RoboDK station: SetToolCutter wrt Tool Holder.rdk

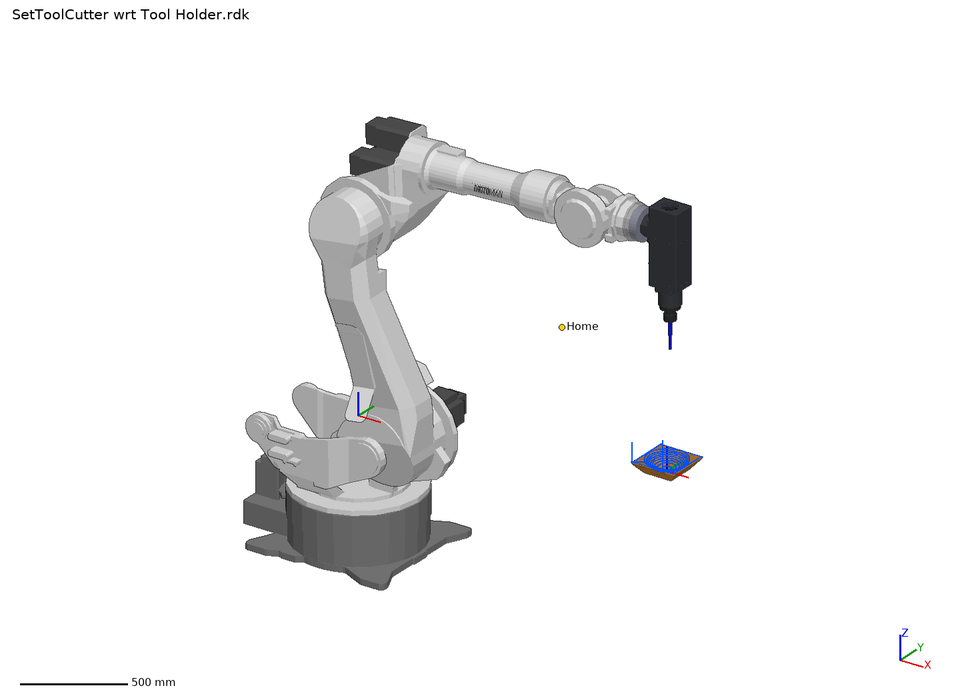
[picture v0: the station drawn from its stored meshes, robots at their saved joint values, targets as dots, program paths as lines]
Station Example Automatic Tool Cutters. Poses are relative to the parent item; angles as X-Y-Z fixed-axis rotations.
  - Python program SetToolCutter (listed below)
  - frame Motoman ES200D Base at (0, 0, 0) mm
    - robot Motoman ES200D: 6 axes, payload 200 kg, reach 2651 mm, repeatability 0.2 mm, weight 1130 kg
        modified DH rows (alpha deg, a mm, theta deg, d mm): 0, 0, 0, 650; -90, 285, -90, 0; 0, 1150, 0, 0; -90, 250, 0, 1225; 90, 0, 0, 0; -90, 0, 0, 250
        base shift (0, 0, -650) mm
        joint limits [-180, -60, -142.5, -360, -125, -360] to [180, 76, 230, 360, 125, 360]; home [0, 0, 0, 0, 0, 0]; saved at [0, -7.655, -4.967, 0, -2.688, 180]
      - tool Tool Holder, TCP at (456.22, 0, 176) mm, rotated rx 0 ry 90 rz 0 deg, size 592.9 x 170 x 256 mm
      - tool Tool 10-150, TCP at (606.22, 0, 176) mm, rotated rx 0 ry 90 rz 0 deg
        - object Cutter 10-150 at (0, 0, 0) mm, size 10 x 10 x 150 mm, geometry from Part.sld
      - tool Tool 20-75, TCP at (531.22, 0, 176) mm, rotated rx 0 ry 90 rz 0 deg
        - object Cutter 20-75 at (0, 0, 0) mm, size 20 x 20 x 75 mm, geometry from Part.sld
    - frame Milling Reference at (1817.19, -92.29, 260.27) mm
      - object Wooden bowl at (0, 0, 0) mm, size 241.3 x 241.3 x 60 mm
      - target Home (joint target) at (-659.05, 92.29, 521.01) mm, rotated rx 180 ry 0 rz -180 deg; joints [0, -37.94, -26.87, 0, -11.07, 180] of Motoman ES200D
  - machining project Machining Settings: Q:/RoboDK/Deploy/RoboDK_vc2013x64/Library/Milling 3axis bowl.nc | rotZ(0) | rotX(0)*rotY(0) | onStart | onPathStart | onApproach | onPoint | onRetract | onFinish | Extruder(%1) | default | default | OutOnMov(%1) | OutOffMov(%1) | onPathFinish | M_RunCode(%1)
  - program Machining (918 instructions, listed below)
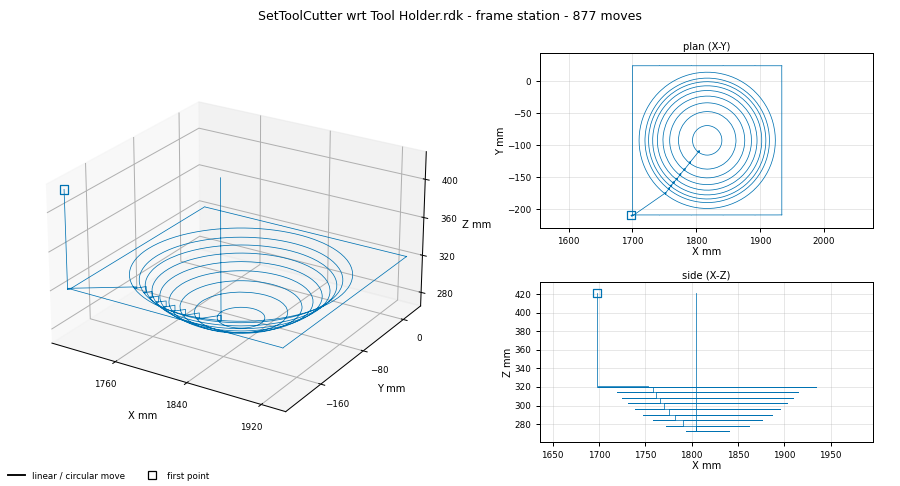
[picture p0: tool path of SetToolCutter wrt Tool Holder.rdk in frame station, 877 of 877 moves have a stored position in this frame; points joined in program order, loops and branches not executed]

--- Python program SetToolCutter ---
# This example shows how to programmatically select (and, if necessary, automatically create) a tool that does not exist
# This is meant to be used for robot machining projects where a tool holder is used as a reference tool
#
# Documentation: https://robodk.com/doc/en/RoboDK-API.html
# Reference:     https://robodk.com/doc/en/PythonAPI/index.html
# Note: It is not required to keep a copy of this file, your python script is saved with the station
from robolink import *    # RoboDK API
from robodk import *      # Robot toolbox
RDK = Robolink()

# Ask the user to select a tool holder
tool_holder = RDK.ItemUserPick('Select a the tool holder (TCP spindle reference)', ITEM_TYPE_TOOL)
# Alernatively, pick a named tool holder:
# tool_holder = RDK.Item('Tool Holder', ITEM_TYPE_TOOL)
# Or, the first tool of a robot:
# tool_holder = robot.Childs()[0]

# Exit if the tool does not exist
if not tool_holder.Valid():
    raise Exception("The tool holder was not selected")

# Retrieve the robot
robot = tool_holder.Parent()

# Ask the user to enter the tool parameters
user_input = mbox("Enter the tool diameter and length (in mm) using the following format:\ndiameter-length\n\nExample:\n10-150", entry="10-150")
if user_input is False:
    print("Operation cancelled")
    quit(0)

# Convert the string to diameter and length variables
diam_length = user_input.split('-')
try:
    diameter = float(diam_length[0])
    length = float(diam_length[1])
except:
    raise Exception("Invalid input: " + diam_length)

# Create a new tool and add the geometry to it
tool_i_name = 'Tool %s' % user_input
tool_i = RDK.Item(tool_i_name, ITEM_TYPE_TOOL)
if tool_i.Valid():
    print("The tool already exists")

else:
    # If the tool holder Z axis points towards the outsite:
    tool_i_pose = tool_holder.PoseTool() * transl(0,0,length)
    # If the tool holder Z axis points towards the inside:
    #tool_i_pose = tool_holder.PoseTool() * transl(0,0,length) * rotx(pi)
    tool_i = robot.AddTool(tool_i_pose, tool_i_name)

    # RoboDK library comes with a sample part that always has the same name
    # this Part.sld is 80 mm in diameter and 100 mm long
    tool1_shape = RDK.AddFile(RDK.getParam('PATH_LIBRARY') + '/Part.sld', tool_i)
    tool1_shape.setName("Cutter %s" % user_input)
    tool1_shape.setGeometryPose(rotx(pi))
    # Scale the object accordingly
    tool1_shape.Scale([ diameter/60,   diameter/60,   length/80  ])
    # Change the color
    tool1_shape.Recolor([0,0,1,0.4]) # make the drill bit blue & transparent (RGBA): if transparency is under 80% it won't check for collisions (when you activate collision checking).


# Set the active tool
robot.setTool(tool_i)

--- program Machining (robot Motoman ES200D) ---
  Set Ref.: Milling Reference
  Set Tool: Tool 10-150
  Show Tool 10-150
  Set speed (1000.0 mm/s)
  Set speed (1000.0 mm/s)
  MoveJ 1 to (-119.55, -117.48, 161.2) mm, rotated rx 180 ry 0 rz 180 deg; joints [-9.367, -12.184, -28.14, -149.033, -18.441, -29.651]
  MoveL 2 to (-119.55, -117.48, 161.2) mm, rotated rx 180 ry 0 rz 180 deg; joints [-9.367, -12.184, -28.14, -149.033, -18.441, -29.651]
  MoveL 3 to (-119.55, -117.48, 61.2) mm, rotated rx -180 ry 0 rz 180 deg; joints [-9.367, -11.562, -32.254, -154.973, -22.628, -23.313]
  MoveL 4 to (-119.55, -117.48, 61.2) mm, rotated rx -180 ry 0 rz 180 deg; joints [-9.367, -11.562, -32.254, -154.973, -22.628, -23.313]
  Set speed (5.0 mm/s)
  MoveL 5 to (-119.55, -117.48, 60) mm, rotated rx -180 ry 0 rz -180 deg; joints [-9.367, -11.552, -32.301, -155.032, -22.68, -23.25]
  MoveL 6 to (-118.15, -118.45, 60) mm, rotated rx -180 ry 0 rz -180 deg; joints [-9.4, -11.471, -32.235, -154.97, -22.707, -23.304]
  MoveL 7 to (-117.59, -118.18, 60) mm, rotated rx -180 ry 0 rz -180 deg; joints [-9.384, -11.444, -32.213, -155.013, -22.705, -23.264]
  MoveL 8 to (-117.24, -117.67, 60) mm, rotated rx -180 ry 0 rz -180 deg; joints [-9.359, -11.43, -32.202, -155.075, -22.698, -23.206]
  MoveL 9 to (-117.19, -117.05, 60) mm, rotated rx -180 ry 0 rz 180 deg; joints [-9.331, -11.433, -32.204, -155.14, -22.686, -23.146]
  Set speed (16.7 mm/s)
  MoveL 10 to (-117.29, -116.49, 60) mm, rotated rx -180 ry 0 rz -180 deg; joints [-9.308, -11.443, -32.212, -155.194, -22.675, -23.096]
  MoveL 11 to (-116.89, -115.89, 60) mm, rotated rx 180 ry 0 rz 180 deg; joints [-9.278, -11.427, -32.2, -155.268, -22.666, -23.028]
  MoveL 12 to (-116.98, -83.97, 60) mm, rotated rx 180 ry 0 rz 180 deg; joints [-7.876, -11.682, -32.407, -158.649, -22.109, -19.909]
  MoveL 13 to (-116.98, 115.67, 60) mm, rotated rx 180 ry 0 rz 180 deg; joints [1.051, -12.311, -32.914, -182.985, -20.629, 2.794]
  MoveL 14 to (-117.29, 116.83, 60) mm, rotated rx 180 ry 0 rz 180 deg; joints [1.103, -12.326, -32.926, -183.133, -20.628, 2.933]
  MoveL 15 to (-117.05, 117.18, 60) mm, rotated rx 180 ry 0 rz 180 deg; joints [1.119, -12.313, -32.916, -183.177, -20.632, 2.974]
  MoveL 16 to (-116.46, 117.29, 60) mm, rotated rx -180 ry 0 rz 180 deg; joints [1.123, -12.282, -32.891, -183.189, -20.638, 2.985]
  MoveL 17 to (-115.99, 116.9, 60) mm, rotated rx -180 ry 0 rz -180 deg; joints [1.106, -12.257, -32.871, -183.137, -20.642, 2.936]
  MoveL 18 to (-110.81, 116.98, 60) mm, rotated rx 180 ry 0 rz 180 deg; joints [1.105, -11.984, -32.651, -183.127, -20.695, 2.926]
  MoveL 19 to (-75.63, 116.98, 60) mm, rotated rx -180 ry 0 rz -180 deg; joints [1.075, -10.139, -31.136, -182.998, -21.023, 2.799]
  MoveL 20 to (-75.08, 117.32, 60) mm, rotated rx 180 ry 0 rz -180 deg; joints [1.09, -10.111, -31.112, -183.038, -21.029, 2.836]
  MoveL 21 to (-74.41, 116.98, 60) mm, rotated rx 180 ry 0 rz 180 deg; joints [1.074, -10.076, -31.083, -182.994, -21.034, 2.795]
  MoveL 22 to (-25.6, 116.98, 60) mm, rotated rx -180 ry 0 rz -180 deg; joints [1.036, -7.548, -28.917, -182.84, -21.392, 2.645]
  MoveL 23 to (-25.06, 117.33, 60) mm, rotated rx -180 ry 0 rz 180 deg; joints [1.05, -7.52, -28.892, -182.879, -21.397, 2.681]
  MoveL 24 to (-24.38, 116.98, 60) mm, rotated rx 180 ry 0 rz 180 deg; joints [1.035, -7.486, -28.862, -182.837, -21.4, 2.642]
  MoveL 25 to (24.43, 116.98, 60) mm, rotated rx -180 ry 0 rz -180 deg; joints [0.999, -4.992, -26.621, -182.709, -21.651, 2.518]
  MoveL 26 to (24.88, 117.31, 60) mm, rotated rx 180 ry 0 rz -180 deg; joints [1.012, -4.969, -26.6, -182.743, -21.654, 2.55]
  MoveL 27 to (25.65, 116.98, 60) mm, rotated rx 180 ry 0 rz 180 deg; joints [0.998, -4.93, -26.564, -182.706, -21.656, 2.515]
  MoveL 28 to (74.35, 116.98, 60) mm, rotated rx 180 ry 0 rz 180 deg; joints [0.965, -2.47, -24.252, -182.599, -21.803, 2.413]
  MoveL 29 to (74.9, 117.32, 60) mm, rotated rx -180 ry 0 rz 180 deg; joints [0.978, -2.442, -24.226, -182.634, -21.805, 2.445]
  MoveL 30 to (75.57, 116.98, 60) mm, rotated rx -180 ry 0 rz -180 deg; joints [0.964, -2.408, -24.193, -182.597, -21.805, 2.411]
  MoveL 31 to (115.94, 116.98, 60) mm, rotated rx 180 ry 0 rz 180 deg; joints [0.938, -0.388, -22.219, -182.522, -21.85, 2.341]
  MoveL 32 to (116.4, 117.29, 60) mm, rotated rx 180 ry 0 rz 180 deg; joints [0.95, -0.365, -22.196, -182.553, -21.851, 2.37]
  MoveL 33 to (116.91, 117.27, 60) mm, rotated rx 180 ry 0 rz 180 deg; joints [0.949, -0.339, -22.171, -182.55, -21.851, 2.367]
  MoveL 34 to (117.31, 116.72, 60) mm, rotated rx -180 ry 0 rz -180 deg; joints [0.928, -0.32, -22.151, -182.494, -21.85, 2.315]
  MoveL 35 to (117.11, 116.16, 60) mm, rotated rx -180 ry 0 rz -180 deg; joints [0.907, -0.33, -22.162, -182.437, -21.849, 2.262]
  MoveL 36 to (116.89, 115.69, 60) mm, rotated rx -180 ry 0 rz -180 deg; joints [0.889, -0.341, -22.173, -182.389, -21.849, 2.218]
  MoveL 37 to (116.98, 83.78, 60) mm, rotated rx 180 ry 0 rz 180 deg; joints [-0.323, -0.345, -22.176, -179.13, -21.834, -0.807]
  MoveL 38 to (116.98, -115.86, 60) mm, rotated rx -180 ry 0 rz -180 deg; joints [-7.858, 0.366, -21.465, -159.638, -23.137, -18.844]
  MoveL 39 to (117.33, -116.64, 60) mm, rotated rx -180 ry 0 rz -180 deg; joints [-7.885, 0.389, -21.443, -159.572, -23.146, -18.905]
  MoveL 40 to (117.02, -117.21, 60) mm, rotated rx -180 ry 0 rz 180 deg; joints [-7.908, 0.378, -21.454, -159.518, -23.153, -18.955]
  MoveL 41 to (116.53, -117.29, 60) mm, rotated rx 180 ry 0 rz 180 deg; joints [-7.914, 0.354, -21.478, -159.505, -23.155, -18.967]
  MoveL 42 to (115.95, -116.9, 60) mm, rotated rx -180 ry 0 rz -180 deg; joints [-7.902, 0.323, -21.509, -159.532, -23.152, -18.942]
  MoveL 43 to (110.78, -116.98, 60) mm, rotated rx -180 ry 0 rz 180 deg; joints [-7.932, 0.068, -21.764, -159.461, -23.162, -19.007]
  MoveL 44 to (75.6, -116.98, 60) mm, rotated rx -180 ry 0 rz -180 deg; joints [-8.12, -1.672, -23.482, -158.992, -23.203, -19.441]
  MoveL 45 to (75.05, -117.33, 60) mm, rotated rx -180 ry 0 rz -180 deg; joints [-8.136, -1.697, -23.506, -158.952, -23.208, -19.478]
  MoveL 46 to (74.38, -116.98, 60) mm, rotated rx -180 ry 0 rz -180 deg; joints [-8.127, -1.733, -23.541, -158.975, -23.203, -19.457]
  MoveL 47 to (25.57, -116.98, 60) mm, rotated rx -180 ry 0 rz -180 deg; joints [-8.403, -4.165, -25.856, -158.216, -23.188, -20.172]
  MoveL 48 to (25.02, -117.34, 60) mm, rotated rx -180 ry 0 rz 180 deg; joints [-8.42, -4.19, -25.879, -158.173, -23.193, -20.211]
  MoveL 49 to (24.35, -116.98, 60) mm, rotated rx -180 ry 0 rz -180 deg; joints [-8.41, -4.226, -25.913, -158.195, -23.187, -20.191]
  MoveL 50 to (-24.36, -116.98, 60) mm, rotated rx -180 ry 0 rz -180 deg; joints [-8.705, -6.679, -28.148, -157.299, -23.089, -21.048]
  MoveL 51 to (-25, -117.35, 60) mm, rotated rx -180 ry 0 rz -180 deg; joints [-8.724, -6.708, -28.174, -157.251, -23.093, -21.092]
  MoveL 52 to (-25.58, -116.98, 60) mm, rotated rx 180 ry 0 rz 180 deg; joints [-8.713, -6.74, -28.203, -157.275, -23.086, -21.071]
  MoveL 53 to (-74.39, -116.98, 60) mm, rotated rx -180 ry 0 rz 180 deg; joints [-9.03, -9.227, -30.367, -156.219, -22.907, -22.093]
  MoveL 54 to (-74.94, -117.33, 60) mm, rotated rx -180 ry 0 rz -180 deg; joints [-9.049, -9.252, -30.388, -156.171, -22.91, -22.137]
  MoveL 55 to (-75.61, -116.98, 60) mm, rotated rx 180 ry 0 rz 180 deg; joints [-9.038, -9.289, -30.42, -156.19, -22.901, -22.121]
  MoveL 56 to (-115.98, -116.98, 60) mm, rotated rx 180 ry 0 rz 180 deg; joints [-9.32, -11.371, -32.154, -155.179, -22.692, -23.108]
  MoveL 57 to (-116.63, -117.33, 60) mm, rotated rx -180 ry 0 rz -180 deg; joints [-9.34, -11.401, -32.179, -155.126, -22.695, -23.158]
  MoveL 58 to (-117.19, -117.05, 60) mm, rotated rx -180 ry 0 rz 180 deg; joints [-9.331, -11.433, -32.204, -155.14, -22.686, -23.146]
  Set speed (16.7 mm/s)
  MoveL 59 to (-117.8, -116.93, 60) mm, rotated rx 180 ry 0 rz 180 deg; joints [-9.33, -11.465, -32.231, -155.136, -22.68, -23.151]
  MoveL 60 to (-118.38, -117.12, 60) mm, rotated rx 180 ry 0 rz 180 deg; joints [-9.343, -11.494, -32.254, -155.1, -22.681, -23.185]
  MoveL 61 to (-118.8, -117.59, 60) mm, rotated rx 180 ry 0 rz -180 deg; joints [-9.367, -11.512, -32.268, -155.041, -22.687, -23.24]
  MoveL 62 to (-118.26, -119.2, 60) mm, rotated rx -180 ry 0 rz -180 deg; joints [-9.433, -11.47, -32.234, -154.89, -22.72, -23.378]
  MoveL 63 to (-118.26, -119.2, 61.2) mm, rotated rx 180 ry 0 rz 180 deg; joints [-9.433, -11.48, -32.187, -154.832, -22.668, -23.441]
  Set speed (1000.0 mm/s)
  MoveL 64 to (-64.77, -81.96, 61.2) mm, rotated rx -180 ry 0 rz 180 deg; joints [-7.484, -9.005, -30.122, -159.967, -22.347, -18.637]
  Set speed (5.0 mm/s)
  MoveL 65 to (-64.77, -81.96, 60) mm, rotated rx 180 ry 0 rz 180 deg; joints [-7.484, -8.994, -30.169, -160.014, -22.401, -18.585]
  MoveL 66 to (-66.46, -82.15, 60) mm, rotated rx 180 ry 0 rz 180 deg; joints [-7.502, -9.08, -30.242, -159.959, -22.395, -18.637]
  MoveL 67 to (-66.71, -82.72, 60) mm, rotated rx -180 ry 0 rz -180 deg; joints [-7.527, -9.088, -30.249, -159.895, -22.402, -18.697]
  MoveL 68 to (-66.64, -83.34, 60) mm, rotated rx 180 ry 0 rz 180 deg; joints [-7.553, -9.08, -30.242, -159.831, -22.411, -18.756]
  MoveL 69 to (-66.26, -83.84, 60) mm, rotated rx -180 ry 0 rz -180 deg; joints [-7.572, -9.058, -30.223, -159.787, -22.42, -18.796]
  Set speed (16.7 mm/s)
  MoveL 70 to (-60.03, -88.41, 60) mm, rotated rx -180 ry 0 rz -180 deg; joints [-7.731, -8.707, -29.922, -159.438, -22.519, -19.112]
  MoveL 71 to (-53.48, -92.52, 60) mm, rotated rx -180 ry 0 rz 180 deg; joints [-7.866, -8.342, -29.608, -159.148, -22.611, -19.373]
  MoveL 72 to (-46.6, -96.17, 60) mm, rotated rx -180 ry 0 rz -180 deg; joints [-7.979, -7.965, -29.281, -158.915, -22.695, -19.582]
  MoveL 73 to (-39.63, -99.24, 60) mm, rotated rx -180 ry 0 rz -180 deg; joints [-8.066, -7.587, -28.951, -158.743, -22.769, -19.733]
  MoveL 74 to (-32.34, -101.86, 60) mm, rotated rx -180 ry 0 rz 180 deg; joints [-8.131, -7.197, -28.607, -158.625, -22.835, -19.835]
  MoveL 75 to (-25.37, -103.8, 60) mm, rotated rx 180 ry 0 rz 180 deg; joints [-8.17, -6.829, -28.281, -158.567, -22.887, -19.883]
  MoveL 76 to (-25.08, -103.7, 60) mm, rotated rx 180 ry 0 rz 180 deg; joints [-8.164, -6.815, -28.269, -158.583, -22.886, -19.868]
  MoveL 77 to (-24.41, -104.03, 60) mm, rotated rx 180 ry 0 rz 180 deg; joints [-8.174, -6.779, -28.237, -158.563, -22.894, -19.886]
  MoveL 78 to (-20.17, -104.94, 60) mm, rotated rx -180 ry 0 rz -180 deg; joints [-8.186, -6.557, -28.039, -158.553, -22.92, -19.891]
  MoveL 79 to (-12.53, -106.13, 60) mm, rotated rx 180 ry 0 rz 180 deg; joints [-8.19, -6.162, -27.685, -158.58, -22.959, -19.861]
  MoveL 80 to (-4.79, -106.76, 60) mm, rotated rx 180 ry 0 rz 180 deg; joints [-8.17, -5.766, -27.328, -158.661, -22.988, -19.781]
  MoveL 81 to (2.85, -106.83, 60) mm, rotated rx -180 ry 0 rz 180 deg; joints [-8.129, -5.38, -26.977, -158.79, -23.007, -19.657]
  MoveL 82 to (10.59, -106.34, 60) mm, rotated rx -180 ry 0 rz 180 deg; joints [-8.065, -4.994, -26.623, -158.972, -23.016, -19.485]
  MoveL 83 to (18.23, -105.3, 60) mm, rotated rx -180 ry 0 rz -180 deg; joints [-7.981, -4.618, -26.276, -159.201, -23.016, -19.27]
  MoveL 84 to (24.4, -104.03, 60) mm, rotated rx -180 ry 0 rz -180 deg; joints [-7.896, -4.317, -25.997, -159.424, -23.008, -19.062]
  MoveL 85 to (24.95, -103.68, 60) mm, rotated rx 180 ry 0 rz 180 deg; joints [-7.879, -4.292, -25.974, -159.466, -23.004, -19.023]
  MoveL 86 to (25.37, -103.8, 60) mm, rotated rx -180 ry 0 rz -180 deg; joints [-7.881, -4.27, -25.953, -159.462, -23.007, -19.027]
  MoveL 87 to (32.05, -101.95, 60) mm, rotated rx -180 ry 0 rz 180 deg; joints [-7.772, -3.948, -25.653, -159.745, -22.991, -18.763]
  MoveL 88 to (39.3, -99.38, 60) mm, rotated rx 180 ry 0 rz 180 deg; joints [-7.631, -3.602, -25.328, -160.102, -22.967, -18.431]
  MoveL 89 to (46.36, -96.29, 60) mm, rotated rx -180 ry 0 rz 180 deg; joints [-7.473, -3.269, -25.015, -160.502, -22.935, -18.061]
  MoveL 90 to (53.22, -92.67, 60) mm, rotated rx 180 ry 0 rz 180 deg; joints [-7.297, -2.95, -24.711, -160.945, -22.896, -17.651]
  MoveL 91 to (59.78, -88.58, 60) mm, rotated rx -180 ry 0 rz -180 deg; joints [-7.106, -2.648, -24.423, -161.426, -22.852, -17.205]
  MoveL 92 to (65.97, -84.07, 60) mm, rotated rx 180 ry 0 rz 180 deg; joints [-6.901, -2.367, -24.154, -161.939, -22.803, -16.731]
  MoveL 93 to (71.86, -79.09, 60) mm, rotated rx -180 ry 0 rz 180 deg; joints [-6.681, -2.103, -23.899, -162.49, -22.75, -16.222]
  MoveL 94 to (74.29, -76.81, 60) mm, rotated rx 180 ry 0 rz 180 deg; joints [-6.582, -1.995, -23.795, -162.739, -22.726, -15.992]
  MoveL 95 to (74.58, -76.19, 60) mm, rotated rx 180 ry 0 rz 180 deg; joints [-6.557, -1.984, -23.784, -162.802, -22.719, -15.934]
  MoveL 96 to (75.15, -75.96, 60) mm, rotated rx -180 ry 0 rz -180 deg; joints [-6.546, -1.957, -23.758, -162.831, -22.717, -15.907]
  MoveL 97 to (80.34, -70.47, 60) mm, rotated rx -180 ry 0 rz 180 deg; joints [-6.312, -1.729, -23.537, -163.42, -22.66, -15.363]
  MoveL 98 to (85.23, -64.46, 60) mm, rotated rx -180 ry 0 rz -180 deg; joints [-6.061, -1.518, -23.332, -164.054, -22.6, -14.777]
  MoveL 99 to (89.66, -58.15, 60) mm, rotated rx 180 ry 0 rz 180 deg; joints [-5.801, -1.33, -23.148, -164.712, -22.54, -14.169]
  MoveL 100 to (93.63, -51.52, 60) mm, rotated rx -180 ry 0 rz 180 deg; joints [-5.532, -1.165, -22.987, -165.396, -22.478, -13.537]
  MoveL 101 to (97.05, -44.73, 60) mm, rotated rx 180 ry 0 rz 180 deg; joints [-5.261, -1.027, -22.851, -166.09, -22.419, -12.896]
  MoveL 102 to (100.02, -37.64, 60) mm, rotated rx -180 ry 0 rz -180 deg; joints [-4.98, -0.911, -22.737, -166.81, -22.359, -12.23]
  MoveL 103 to (102.44, -30.41, 60) mm, rotated rx 180 ry 0 rz 180 deg; joints [-4.696, -0.82, -22.647, -167.541, -22.302, -11.553]
  MoveL 104 to (102.51, -30.2, 60) mm, rotated rx -180 ry 0 rz -180 deg; joints [-4.688, -0.818, -22.645, -167.562, -22.301, -11.533]
  MoveL 105 to (104.4, -22.82, 60) mm, rotated rx -180 ry 0 rz 180 deg; joints [-4.401, -0.753, -22.581, -168.305, -22.246, -10.846]
  MoveL 106 to (105.76, -15.32, 60) mm, rotated rx 180 ry 0 rz 180 deg; joints [-4.112, -0.713, -22.541, -169.058, -22.194, -10.149]
  MoveL 107 to (106.59, -7.67, 60) mm, rotated rx -180 ry 0 rz -180 deg; joints [-3.818, -0.698, -22.527, -169.824, -22.144, -9.439]
  MoveL 108 to (106.86, -0.29, 60) mm, rotated rx -180 ry 0 rz 180 deg; joints [-3.536, -0.709, -22.537, -170.563, -22.099, -8.755]
  MoveL 109 to (106.86, 0.23, 60) mm, rotated rx 180 ry 0 rz 180 deg; joints [-3.517, -0.71, -22.538, -170.615, -22.096, -8.706]
  MoveL 110 to (106.57, 7.9, 60) mm, rotated rx 180 ry 0 rz 180 deg; joints [-3.225, -0.747, -22.575, -171.383, -22.053, -7.995]
  MoveL 111 to (105.8, 14.83, 60) mm, rotated rx 180 ry 0 rz 180 deg; joints [-2.962, -0.804, -22.631, -172.077, -22.017, -7.352]
  MoveL 112 to (104.08, 24.16, 60) mm, rotated rx 180 ry 0 rz 180 deg; joints [-2.609, -0.913, -22.738, -173.013, -21.973, -6.484]
  MoveL 113 to (102.39, 30.57, 60) mm, rotated rx 180 ry 0 rz 180 deg; joints [-2.367, -1.011, -22.835, -173.656, -21.946, -5.887]
  MoveL 114 to (102.13, 31.4, 60) mm, rotated rx 180 ry 0 rz 180 deg; joints [-2.335, -1.026, -22.849, -173.741, -21.942, -5.809]
  MoveL 115 to (99.93, 37.84, 60) mm, rotated rx -180 ry 0 rz -180 deg; joints [-2.091, -1.148, -22.97, -174.389, -21.917, -5.208]
  MoveL 116 to (99.72, 38.39, 60) mm, rotated rx -180 ry 0 rz 180 deg; joints [-2.07, -1.159, -22.981, -174.445, -21.915, -5.156]
  MoveL 117 to (96.85, 45.16, 60) mm, rotated rx -180 ry 0 rz -180 deg; joints [-1.814, -1.314, -23.133, -175.129, -21.89, -4.521]
  MoveL 118 to (96.68, 45.51, 60) mm, rotated rx 180 ry 0 rz 180 deg; joints [-1.801, -1.323, -23.141, -175.164, -21.889, -4.489]
  MoveL 119 to (93.35, 52.01, 60) mm, rotated rx -180 ry 0 rz 180 deg; joints [-1.554, -1.5, -23.314, -175.824, -21.867, -3.877]
  MoveL 120 to (93.2, 52.28, 60) mm, rotated rx 180 ry 0 rz 180 deg; joints [-1.544, -1.508, -23.322, -175.851, -21.866, -3.851]
  MoveL 121 to (89.26, 58.76, 60) mm, rotated rx 180 ry 0 rz 180 deg; joints [-1.297, -1.713, -23.522, -176.511, -21.845, -3.239]
  MoveL 122 to (84.86, 64.95, 60) mm, rotated rx 180 ry 0 rz 180 deg; joints [-1.061, -1.94, -23.741, -177.145, -21.826, -2.651]
  MoveL 123 to (80.02, 70.83, 60) mm, rotated rx 180 ry 0 rz 180 deg; joints [-0.836, -2.188, -23.981, -177.75, -21.809, -2.089]
  MoveL 124 to (79.89, 70.98, 60) mm, rotated rx 180 ry 0 rz 180 deg; joints [-0.83, -2.194, -23.988, -177.765, -21.808, -2.075]
  MoveL 125 to (75.22, 75.88, 60) mm, rotated rx 180 ry 0 rz 180 deg; joints [-0.641, -2.432, -24.216, -178.273, -21.793, -1.604]
  MoveL 126 to (74.66, 76.14, 60) mm, rotated rx 180 ry 0 rz 180 deg; joints [-0.631, -2.46, -24.243, -178.3, -21.792, -1.579]
  MoveL 127 to (74.23, 76.87, 60) mm, rotated rx -180 ry 0 rz -180 deg; joints [-0.603, -2.482, -24.265, -178.375, -21.79, -1.509]
  MoveL 128 to (72.13, 78.85, 60) mm, rotated rx 180 ry 0 rz 180 deg; joints [-0.526, -2.589, -24.366, -178.582, -21.784, -1.317]
  MoveL 129 to (66.22, 83.87, 60) mm, rotated rx -180 ry 0 rz 180 deg; joints [-0.331, -2.888, -24.652, -179.108, -21.767, -0.829]
  MoveL 130 to (59.99, 88.44, 60) mm, rotated rx 180 ry 0 rz 180 deg; joints [-0.152, -3.203, -24.952, -179.589, -21.749, -0.381]
  MoveL 131 to (53.44, 92.54, 60) mm, rotated rx -180 ry 0 rz -180 deg; joints [0.01, -3.534, -25.264, -180.027, -21.731, 0.025]
  MoveL 132 to (46.68, 96.13, 60) mm, rotated rx 180 ry 0 rz 180 deg; joints [0.153, -3.875, -25.585, -180.414, -21.711, 0.384]
  MoveL 133 to (39.59, 99.26, 60) mm, rotated rx 180 ry 0 rz -180 deg; joints [0.279, -4.233, -25.919, -180.755, -21.688, 0.702]
  MoveL 134 to (32.3, 101.87, 60) mm, rotated rx 180 ry 0 rz -180 deg; joints [0.385, -4.602, -26.261, -181.044, -21.663, 0.97]
  MoveL 135 to (25.33, 103.81, 60) mm, rotated rx 180 ry 0 rz -180 deg; joints [0.466, -4.954, -26.587, -181.263, -21.637, 1.174]
  MoveL 136 to (25.05, 103.68, 60) mm, rotated rx -180 ry 0 rz -180 deg; joints [0.461, -4.969, -26.6, -181.25, -21.636, 1.162]
  MoveL 137 to (24.5, 103.91, 60) mm, rotated rx -180 ry 0 rz -180 deg; joints [0.47, -4.997, -26.626, -181.276, -21.634, 1.186]
  MoveL 138 to (20.14, 104.95, 60) mm, rotated rx 180 ry 0 rz 180 deg; joints [0.514, -5.218, -26.828, -181.395, -21.616, 1.297]
  MoveL 139 to (12.5, 106.13, 60) mm, rotated rx 180 ry 0 rz 180 deg; joints [0.565, -5.606, -27.183, -181.536, -21.583, 1.428]
  MoveL 140 to (4.86, 106.75, 60) mm, rotated rx 180 ry 0 rz 180 deg; joints [0.594, -5.995, -27.535, -181.616, -21.547, 1.503]
  MoveL 141 to (-2.88, 106.83, 60) mm, rotated rx 180 ry 0 rz 180 deg; joints [0.6, -6.391, -27.891, -181.636, -21.508, 1.522]
  MoveL 142 to (-10.62, 106.34, 60) mm, rotated rx 180 ry 0 rz 180 deg; joints [0.583, -6.787, -28.245, -181.593, -21.465, 1.482]
  MoveL 143 to (-18.26, 105.29, 60) mm, rotated rx 180 ry 0 rz -180 deg; joints [0.543, -7.18, -28.592, -181.486, -21.419, 1.383]
  MoveL 144 to (-24.43, 104.02, 60) mm, rotated rx 180 ry 0 rz 180 deg; joints [0.492, -7.497, -28.872, -181.349, -21.38, 1.256]
  MoveL 145 to (-24.98, 103.67, 60) mm, rotated rx 180 ry 0 rz 180 deg; joints [0.477, -7.525, -28.897, -181.309, -21.376, 1.219]
  MoveL 146 to (-25.31, 103.82, 60) mm, rotated rx -180 ry 0 rz -180 deg; joints [0.483, -7.542, -28.912, -181.326, -21.375, 1.235]
  MoveL 147 to (-31.99, 101.96, 60) mm, rotated rx 180 ry 0 rz 180 deg; joints [0.408, -7.887, -29.213, -181.121, -21.33, 1.044]
  MoveL 148 to (-39.34, 99.36, 60) mm, rotated rx -180 ry 0 rz -180 deg; joints [0.3, -8.267, -29.543, -180.826, -21.278, 0.77]
  MoveL 149 to (-46.39, 96.27, 60) mm, rotated rx 180 ry 0 rz 180 deg; joints [0.17, -8.632, -29.858, -180.468, -21.227, 0.436]
  MoveL 150 to (-53.25, 92.65, 60) mm, rotated rx 180 ry 0 rz 180 deg; joints [0.015, -8.988, -30.163, -180.043, -21.175, 0.04]
  MoveL 151 to (-59.72, 88.62, 60) mm, rotated rx -180 ry 0 rz 180 deg; joints [-0.158, -9.323, -30.449, -179.561, -21.126, -0.409]
  MoveL 152 to (-66, 84.05, 60) mm, rotated rx 180 ry 0 rz 180 deg; joints [-0.356, -9.648, -30.724, -179.009, -21.079, -0.925]
  MoveL 153 to (-71.9, 79.07, 60) mm, rotated rx 180 ry 0 rz 180 deg; joints [-0.574, -9.953, -30.98, -178.4, -21.035, -1.494]
  MoveL 154 to (-74.23, 76.86, 60) mm, rotated rx -180 ry 0 rz -180 deg; joints [-0.671, -10.074, -31.082, -178.128, -21.018, -1.748]
  MoveL 155 to (-74.45, 76.38, 60) mm, rotated rx 180 ry 0 rz 180 deg; joints [-0.693, -10.085, -31.091, -178.069, -21.017, -1.803]
  MoveL 156 to (-75.18, 75.93, 60) mm, rotated rx 180 ry 0 rz 180 deg; joints [-0.712, -10.123, -31.122, -178.013, -21.011, -1.855]
  MoveL 157 to (-80.37, 70.43, 60) mm, rotated rx 180 ry 0 rz 180 deg; joints [-0.955, -10.389, -31.345, -177.33, -20.976, -2.493]
  MoveL 158 to (-85.26, 64.42, 60) mm, rotated rx 180 ry 0 rz 180 deg; joints [-1.222, -10.639, -31.552, -176.579, -20.947, -3.196]
  MoveL 159 to (-89.69, 58.1, 60) mm, rotated rx 180 ry 0 rz 180 deg; joints [-1.505, -10.863, -31.737, -175.783, -20.926, -3.939]
  MoveL 160 to (-93.58, 51.61, 60) mm, rotated rx -180 ry 0 rz -180 deg; joints [-1.796, -11.057, -31.896, -174.964, -20.913, -4.706]
  MoveL 161 to (-97.08, 44.68, 60) mm, rotated rx -180 ry 0 rz 180 deg; joints [-2.107, -11.228, -32.037, -174.087, -20.911, -5.526]
  MoveL 162 to (-100.04, 37.58, 60) mm, rotated rx -180 ry 0 rz 180 deg; joints [-2.426, -11.369, -32.152, -173.19, -20.918, -6.365]
  MoveL 163 to (-102.47, 30.34, 60) mm, rotated rx 180 ry 0 rz 180 deg; joints [-2.752, -11.479, -32.242, -172.278, -20.936, -7.218]
  MoveL 164 to (-104.36, 22.98, 60) mm, rotated rx -180 ry 0 rz 180 deg; joints [-3.083, -11.559, -32.307, -171.354, -20.966, -8.081]
  MoveL 165 to (-104.42, 22.72, 60) mm, rotated rx -180 ry 0 rz 180 deg; joints [-3.095, -11.561, -32.308, -171.322, -20.967, -8.111]
  MoveL 166 to (-105.73, 15.5, 60) mm, rotated rx 180 ry 0 rz 180 deg; joints [-3.419, -11.608, -32.347, -170.424, -21.006, -8.95]
  MoveL 167 to (-105.78, 15.2, 60) mm, rotated rx -180 ry 0 rz 180 deg; joints [-3.432, -11.61, -32.348, -170.386, -21.008, -8.985]
  MoveL 168 to (-106.57, 7.9, 60) mm, rotated rx -180 ry 0 rz 180 deg; joints [-3.759, -11.627, -32.362, -169.488, -21.058, -9.824]
  MoveL 169 to (-106.6, 7.51, 60) mm, rotated rx 180 ry 0 rz 180 deg; joints [-3.776, -11.627, -32.362, -169.441, -21.061, -9.868]
  MoveL 170 to (-106.86, 0.13, 60) mm, rotated rx 180 ry 0 rz 180 deg; joints [-4.105, -11.615, -32.352, -168.543, -21.122, -10.705]
  MoveL 171 to (-106.86, -0.45, 60) mm, rotated rx -180 ry 0 rz -180 deg; joints [-4.13, -11.612, -32.35, -168.474, -21.127, -10.77]
  MoveL 172 to (-106.55, -8.18, 60) mm, rotated rx 180 ry 0 rz 180 deg; joints [-4.472, -11.566, -32.312, -167.549, -21.202, -11.632]
  MoveL 173 to (-105.74, -15.34, 60) mm, rotated rx -180 ry 0 rz 180 deg; joints [-4.786, -11.493, -32.253, -166.709, -21.281, -12.414]
  MoveL 174 to (-104.19, -23.72, 60) mm, rotated rx -180 ry 0 rz -180 deg; joints [-5.151, -11.374, -32.156, -165.746, -21.384, -13.309]
  MoveL 175 to (-102.5, -30.12, 60) mm, rotated rx 180 ry 0 rz -180 deg; joints [-5.426, -11.254, -32.058, -165.026, -21.47, -13.977]
  MoveL 176 to (-102.21, -31.18, 60) mm, rotated rx 180 ry 0 rz 180 deg; joints [-5.472, -11.234, -32.041, -164.909, -21.484, -14.086]
  MoveL 177 to (-99.79, -38.25, 60) mm, rotated rx 180 ry 0 rz 180 deg; joints [-5.772, -11.071, -31.908, -164.136, -21.588, -14.802]
  MoveL 178 to (-96.91, -45.01, 60) mm, rotated rx -180 ry 0 rz 180 deg; joints [-6.056, -10.884, -31.755, -163.417, -21.693, -15.466]
  MoveL 179 to (-96.74, -45.4, 60) mm, rotated rx -180 ry 0 rz -180 deg; joints [-6.072, -10.873, -31.745, -163.377, -21.7, -15.504]
  MoveL 180 to (-93.25, -52.2, 60) mm, rotated rx -180 ry 0 rz 180 deg; joints [-6.352, -10.653, -31.564, -162.677, -21.813, -16.15]
  MoveL 181 to (-89.31, -58.69, 60) mm, rotated rx -180 ry 0 rz -180 deg; joints [-6.615, -10.41, -31.362, -162.031, -21.927, -16.745]
  MoveL 182 to (-84.91, -64.88, 60) mm, rotated rx -180 ry 0 rz -180 deg; joints [-6.861, -10.144, -31.14, -161.437, -22.041, -17.29]
  MoveL 183 to (-84.78, -65.06, 60) mm, rotated rx 180 ry 0 rz 180 deg; joints [-6.868, -10.136, -31.133, -161.421, -22.044, -17.305]
  MoveL 184 to (-79.93, -70.93, 60) mm, rotated rx 180 ry 0 rz 180 deg; joints [-7.096, -9.848, -30.892, -160.881, -22.157, -17.799]
  MoveL 185 to (-75.14, -75.97, 60) mm, rotated rx 180 ry 0 rz 180 deg; joints [-7.286, -9.568, -30.656, -160.438, -22.257, -18.205]
  MoveL 186 to (-74.59, -76.19, 60) mm, rotated rx -180 ry 0 rz -180 deg; joints [-7.292, -9.538, -30.631, -160.425, -22.263, -18.215]
  MoveL 187 to (-74.27, -76.83, 60) mm, rotated rx -180 ry 0 rz -180 deg; joints [-7.318, -9.517, -30.613, -160.364, -22.274, -18.272]
  MoveL 188 to (-72.17, -78.81, 60) mm, rotated rx -180 ry 0 rz -180 deg; joints [-7.391, -9.396, -30.511, -160.196, -22.315, -18.425]
  MoveL 189 to (-66.26, -83.84, 60) mm, rotated rx -180 ry 0 rz -180 deg; joints [-7.572, -9.058, -30.223, -159.787, -22.42, -18.796]
  Set speed (16.7 mm/s)
  MoveL 190 to (-65.69, -84.09, 60) mm, rotated rx -180 ry 0 rz -180 deg; joints [-7.58, -9.027, -30.197, -159.773, -22.427, -18.809]
  MoveL 191 to (-65.08, -84.01, 60) mm, rotated rx -180 ry 0 rz 180 deg; joints [-7.573, -8.996, -30.17, -159.793, -22.429, -18.79]
  MoveL 192 to (-64.58, -83.64, 60) mm, rotated rx -180 ry 0 rz 180 deg; joints [-7.554, -8.973, -30.15, -159.842, -22.426, -18.744]
  MoveL 193 to (-64.78, -81.95, 60) mm, rotated rx -180 ry 0 rz 180 deg; joints [-7.484, -8.994, -30.169, -160.014, -22.401, -18.585]
  MoveL 194 to (-59.1, -74.54, 60) mm, rotated rx -180 ry 0 rz 180 deg; joints [-7.139, -8.752, -29.961, -160.905, -22.326, -17.757]
  Set speed (5.0 mm/s)
  MoveL 195 to (-59.1, -74.54, 54) mm, rotated rx 180 ry 0 rz 180 deg; joints [-7.139, -8.698, -30.194, -161.131, -22.597, -17.512]
  MoveL 196 to (-60.79, -74.76, 54) mm, rotated rx -180 ry 0 rz -180 deg; joints [-7.157, -8.783, -30.267, -161.076, -22.591, -17.565]
  MoveL 197 to (-61.03, -75.33, 54) mm, rotated rx -180 ry 0 rz -180 deg; joints [-7.182, -8.792, -30.274, -161.012, -22.598, -17.624]
  MoveL 198 to (-60.95, -75.95, 54) mm, rotated rx 180 ry 0 rz 180 deg; joints [-7.208, -8.784, -30.267, -160.949, -22.606, -17.682]
  MoveL 199 to (-60.57, -76.44, 54) mm, rotated rx -180 ry 0 rz -180 deg; joints [-7.227, -8.761, -30.248, -160.905, -22.615, -17.722]
  Set speed (16.7 mm/s)
  MoveL 200 to (-56.23, -79.78, 54) mm, rotated rx -180 ry 0 rz 180 deg; joints [-7.345, -8.516, -30.038, -160.641, -22.684, -17.962]
  MoveL 201 to (-50.68, -83.42, 54) mm, rotated rx 180 ry 0 rz 180 deg; joints [-7.468, -8.208, -29.771, -160.371, -22.761, -18.205]
  MoveL 202 to (-47.04, -85.53, 54) mm, rotated rx 180 ry 0 rz 180 deg; joints [-7.536, -8.007, -29.597, -160.225, -22.808, -18.336]
  MoveL 203 to (-42.43, -87.91, 54) mm, rotated rx -180 ry 0 rz 180 deg; joints [-7.61, -7.755, -29.377, -160.07, -22.861, -18.474]
  MoveL 204 to (-38.66, -89.63, 54) mm, rotated rx -180 ry 0 rz 180 deg; joints [-7.661, -7.551, -29.198, -159.967, -22.901, -18.566]
  MoveL 205 to (-33.94, -91.52, 54) mm, rotated rx -180 ry 0 rz -180 deg; joints [-7.713, -7.297, -28.975, -159.865, -22.947, -18.656]
  MoveL 206 to (-27.98, -93.52, 54) mm, rotated rx 180 ry 0 rz 180 deg; joints [-7.762, -6.98, -28.695, -159.777, -22.997, -18.733]
  MoveL 207 to (-23.49, -94.68, 54) mm, rotated rx -180 ry 0 rz 180 deg; joints [-7.784, -6.744, -28.485, -159.743, -23.029, -18.76]
  MoveL 208 to (-17.44, -96.04, 54) mm, rotated rx -180 ry 0 rz 180 deg; joints [-7.806, -6.427, -28.203, -159.718, -23.068, -18.779]
  MoveL 209 to (-10.76, -97.01, 54) mm, rotated rx 180 ry 0 rz 180 deg; joints [-7.808, -6.082, -27.892, -159.741, -23.102, -18.752]
  MoveL 210 to (-3.33, -97.55, 54) mm, rotated rx 180 ry 0 rz 180 deg; joints [-7.789, -5.703, -27.55, -159.817, -23.13, -18.678]
  MoveL 211 to (4.18, -97.52, 54) mm, rotated rx -180 ry 0 rz -180 deg; joints [-7.746, -5.324, -27.204, -159.947, -23.148, -18.553]
  MoveL 212 to (12, -96.87, 54) mm, rotated rx 180 ry 0 rz 180 deg; joints [-7.678, -4.934, -26.848, -160.139, -23.157, -18.372]
  MoveL 213 to (19.6, -95.62, 54) mm, rotated rx -180 ry 0 rz -180 deg; joints [-7.587, -4.56, -26.503, -160.381, -23.156, -18.146]
  MoveL 214 to (25.63, -94.19, 54) mm, rotated rx 180 ry 0 rz 180 deg; joints [-7.498, -4.266, -26.23, -160.613, -23.148, -17.93]
  MoveL 215 to (32.84, -91.92, 54) mm, rotated rx -180 ry 0 rz -180 deg; joints [-7.371, -3.919, -25.906, -160.939, -23.131, -17.627]
  MoveL 216 to (39.66, -89.19, 54) mm, rotated rx -180 ry 0 rz -180 deg; joints [-7.229, -3.595, -25.602, -161.3, -23.107, -17.293]
  MoveL 217 to (45.82, -86.19, 54) mm, rotated rx 180 ry 0 rz 180 deg; joints [-7.08, -3.306, -25.328, -161.673, -23.079, -16.947]
  MoveL 218 to (51.7, -82.78, 54) mm, rotated rx -180 ry 0 rz -180 deg; joints [-6.918, -3.032, -25.069, -162.079, -23.046, -16.572]
  MoveL 219 to (58.29, -78.29, 54) mm, rotated rx -180 ry 0 rz 180 deg; joints [-6.712, -2.729, -24.781, -162.595, -23.001, -16.095]
  MoveL 220 to (64.31, -73.43, 54) mm, rotated rx 180 ry 0 rz 180 deg; joints [-6.496, -2.457, -24.52, -163.137, -22.953, -15.596]
  MoveL 221 to (70.02, -68, 54) mm, rotated rx -180 ry 0 rz -180 deg; joints [-6.26, -2.202, -24.274, -163.726, -22.9, -15.052]
  MoveL 222 to (73.58, -64.14, 54) mm, rotated rx 180 ry 0 rz 180 deg; joints [-6.096, -2.045, -24.123, -164.138, -22.863, -14.671]
  MoveL 223 to (78.46, -58.07, 54) mm, rotated rx -180 ry 0 rz 180 deg; joints [-5.842, -1.833, -23.918, -164.777, -22.807, -14.082]
  MoveL 224 to (82.62, -51.96, 54) mm, rotated rx 180 ry 0 rz 180 deg; joints [-5.59, -1.656, -23.746, -165.411, -22.752, -13.497]
  MoveL 225 to (85.72, -46.69, 54) mm, rotated rx 180 ry 0 rz 180 deg; joints [-5.376, -1.527, -23.62, -165.953, -22.706, -12.997]
  MoveL 226 to (88.55, -41.08, 54) mm, rotated rx -180 ry 0 rz -180 deg; joints [-5.15, -1.412, -23.508, -166.525, -22.659, -12.468]
  MoveL 227 to (90.89, -35.55, 54) mm, rotated rx 180 ry 0 rz 180 deg; joints [-4.93, -1.32, -23.417, -167.085, -22.614, -11.952]
  MoveL 228 to (93.41, -28.31, 54) mm, rotated rx -180 ry 0 rz -180 deg; joints [-4.644, -1.224, -23.324, -167.815, -22.559, -11.277]
  MoveL 229 to (95.7, -19.21, 54) mm, rotated rx -180 ry 0 rz -180 deg; joints [-4.288, -1.145, -23.246, -168.728, -22.493, -10.434]
  MoveL 230 to (96.89, -11.85, 54) mm, rotated rx -180 ry 0 rz -180 deg; joints [-4.003, -1.113, -23.215, -169.463, -22.444, -9.755]
  MoveL 231 to (97.24, -8.25, 54) mm, rotated rx 180 ry 0 rz 180 deg; joints [-3.864, -1.107, -23.209, -169.822, -22.421, -9.423]
  MoveL 232 to (97.61, 0.22, 54) mm, rotated rx 180 ry 0 rz 180 deg; joints [-3.539, -1.116, -23.218, -170.666, -22.369, -8.643]
  MoveL 233 to (97.35, 7.15, 54) mm, rotated rx -180 ry 0 rz -180 deg; joints [-3.274, -1.15, -23.251, -171.356, -22.33, -8.005]
  MoveL 234 to (96.62, 13.85, 54) mm, rotated rx -180 ry 0 rz -180 deg; joints [-3.018, -1.205, -23.305, -172.023, -22.295, -7.388]
  MoveL 235 to (95.2, 21.54, 54) mm, rotated rx 180 ry 0 rz 180 deg; joints [-2.725, -1.295, -23.393, -172.789, -22.257, -6.679]
  MoveL 236 to (94.39, 24.84, 54) mm, rotated rx -180 ry 0 rz 180 deg; joints [-2.6, -1.343, -23.44, -173.118, -22.242, -6.374]
  MoveL 237 to (92.09, 32.36, 54) mm, rotated rx 180 ry 0 rz 180 deg; joints [-2.314, -1.474, -23.568, -173.868, -22.209, -5.68]
  MoveL 238 to (88.9, 40.32, 54) mm, rotated rx 180 ry 0 rz 180 deg; joints [-2.011, -1.649, -23.739, -174.665, -22.177, -4.942]
  MoveL 239 to (86.15, 45.85, 54) mm, rotated rx 180 ry 0 rz 180 deg; joints [-1.801, -1.796, -23.882, -175.221, -22.155, -4.428]
  MoveL 240 to (82.85, 51.62, 54) mm, rotated rx -180 ry 0 rz 180 deg; joints [-1.581, -1.97, -24.05, -175.801, -22.134, -3.89]
  MoveL 241 to (77.98, 58.71, 54) mm, rotated rx 180 ry 0 rz 180 deg; joints [-1.309, -2.223, -24.295, -176.519, -22.109, -3.225]
  MoveL 242 to (74.02, 63.62, 54) mm, rotated rx -180 ry 0 rz 180 deg; joints [-1.121, -2.427, -24.491, -177.018, -22.091, -2.763]
  MoveL 243 to (69.32, 68.72, 54) mm, rotated rx 180 ry 0 rz 180 deg; joints [-0.925, -2.668, -24.722, -177.539, -22.072, -2.281]
  MoveL 244 to (62.83, 74.7, 54) mm, rotated rx -180 ry 0 rz 180 deg; joints [-0.693, -2.999, -25.038, -178.153, -22.049, -1.712]
  MoveL 245 to (56.19, 79.8, 54) mm, rotated rx 180 ry 0 rz 180 deg; joints [-0.494, -3.337, -25.358, -178.682, -22.026, -1.222]
  MoveL 246 to (50.64, 83.45, 54) mm, rotated rx -180 ry 0 rz -180 deg; joints [-0.352, -3.618, -25.623, -179.062, -22.008, -0.87]
  MoveL 247 to (47, 85.55, 54) mm, rotated rx 180 ry 0 rz 180 deg; joints [-0.269, -3.803, -25.797, -179.283, -21.996, -0.665]
  MoveL 248 to (42.39, 87.93, 54) mm, rotated rx 180 ry 0 rz 180 deg; joints [-0.175, -4.036, -26.015, -179.534, -21.98, -0.432]
  MoveL 249 to (38.62, 89.65, 54) mm, rotated rx -180 ry 0 rz 180 deg; joints [-0.106, -4.228, -26.194, -179.717, -21.966, -0.263]
  MoveL 250 to (34.01, 91.49, 54) mm, rotated rx 180 ry 0 rz 180 deg; joints [-0.032, -4.461, -26.411, -179.914, -21.95, -0.08]
  MoveL 251 to (27.94, 93.53, 54) mm, rotated rx 180 ry 0 rz 180 deg; joints [0.05, -4.769, -26.696, -180.134, -21.927, 0.124]
  MoveL 252 to (23.66, 94.66, 54) mm, rotated rx -180 ry 0 rz -180 deg; joints [0.096, -4.986, -26.896, -180.257, -21.909, 0.238]
  MoveL 253 to (17.41, 96.05, 54) mm, rotated rx -180 ry 0 rz -180 deg; joints [0.153, -5.304, -27.187, -180.41, -21.883, 0.38]
  MoveL 254 to (10.72, 97.02, 54) mm, rotated rx 180 ry 0 rz -180 deg; joints [0.193, -5.645, -27.497, -180.519, -21.853, 0.481]
  MoveL 255 to (3.3, 97.56, 54) mm, rotated rx 180 ry 0 rz 180 deg; joints [0.216, -6.023, -27.84, -180.582, -21.817, 0.54]
  MoveL 256 to (-4.22, 97.52, 54) mm, rotated rx 180 ry 0 rz 180 deg; joints [0.216, -6.408, -28.185, -180.582, -21.778, 0.541]
  MoveL 257 to (-12.03, 96.87, 54) mm, rotated rx 180 ry 0 rz 180 deg; joints [0.19, -6.808, -28.542, -180.513, -21.735, 0.477]
  MoveL 258 to (-19.63, 95.62, 54) mm, rotated rx 180 ry 0 rz -180 deg; joints [0.139, -7.198, -28.888, -180.376, -21.69, 0.349]
  MoveL 259 to (-25.67, 94.18, 54) mm, rotated rx -180 ry 0 rz 180 deg; joints [0.079, -7.509, -29.162, -180.214, -21.653, 0.199]
  MoveL 260 to (-32.78, 91.94, 54) mm, rotated rx -180 ry 0 rz 180 deg; joints [-0.015, -7.875, -29.482, -179.96, -21.607, -0.037]
  MoveL 261 to (-39.6, 89.22, 54) mm, rotated rx -180 ry 0 rz -180 deg; joints [-0.13, -8.227, -29.788, -179.645, -21.561, -0.33]
  MoveL 262 to (-45.76, 86.22, 54) mm, rotated rx 180 ry 0 rz 180 deg; joints [-0.259, -8.545, -30.063, -179.295, -21.519, -0.656]
  MoveL 263 to (-51.73, 82.77, 54) mm, rotated rx -180 ry 0 rz -180 deg; joints [-0.408, -8.853, -30.327, -178.887, -21.478, -1.036]
  MoveL 264 to (-57.7, 78.73, 54) mm, rotated rx -180 ry 0 rz -180 deg; joints [-0.583, -9.161, -30.59, -178.406, -21.436, -1.484]
  MoveL 265 to (-63.11, 74.46, 54) mm, rotated rx -180 ry 0 rz 180 deg; joints [-0.769, -9.44, -30.827, -177.891, -21.4, -1.964]
  MoveL 266 to (-67.3, 70.67, 54) mm, rotated rx 180 ry 0 rz 180 deg; joints [-0.936, -9.655, -31.008, -177.431, -21.373, -2.392]
  MoveL 267 to (-72.52, 65.34, 54) mm, rotated rx -180 ry 0 rz -180 deg; joints [-1.171, -9.922, -31.233, -176.781, -21.342, -2.999]
  MoveL 268 to (-77.18, 59.76, 54) mm, rotated rx 180 ry 0 rz 180 deg; joints [-1.418, -10.158, -31.431, -176.096, -21.318, -3.638]
  MoveL 269 to (-80.75, 54.84, 54) mm, rotated rx -180 ry 0 rz -180 deg; joints [-1.637, -10.338, -31.581, -175.49, -21.303, -4.203]
  MoveL 270 to (-84.21, 49.36, 54) mm, rotated rx -180 ry 0 rz 180 deg; joints [-1.881, -10.51, -31.724, -174.813, -21.293, -4.835]
  MoveL 271 to (-87.25, 43.77, 54) mm, rotated rx 180 ry 0 rz 180 deg; joints [-2.131, -10.659, -31.847, -174.121, -21.29, -5.48]
  MoveL 272 to (-90.08, 37.6, 54) mm, rotated rx -180 ry 0 rz -180 deg; joints [-2.407, -10.794, -31.959, -173.359, -21.295, -6.191]
  MoveL 273 to (-92.86, 30.08, 54) mm, rotated rx -180 ry 0 rz -180 deg; joints [-2.743, -10.922, -32.064, -172.433, -21.312, -7.055]
  MoveL 274 to (-94.35, 24.94, 54) mm, rotated rx 180 ry 0 rz 180 deg; joints [-2.973, -10.987, -32.118, -171.801, -21.33, -7.644]
  MoveL 275 to (-95.72, 19.11, 54) mm, rotated rx 180 ry 0 rz 180 deg; joints [-3.233, -11.042, -32.163, -171.09, -21.356, -8.307]
  MoveL 276 to (-96.9, 11.74, 54) mm, rotated rx -180 ry 0 rz 180 deg; joints [-3.561, -11.081, -32.195, -170.198, -21.399, -9.138]
  MoveL 277 to (-97.57, 2.67, 54) mm, rotated rx -180 ry 0 rz 180 deg; joints [-3.963, -11.085, -32.198, -169.113, -21.465, -10.148]
  MoveL 278 to (-97.61, -0.98, 54) mm, rotated rx -180 ry 0 rz -180 deg; joints [-4.124, -11.073, -32.189, -168.681, -21.496, -10.55]
  MoveL 279 to (-97.32, -7.49, 54) mm, rotated rx 180 ry 0 rz 180 deg; joints [-4.41, -11.033, -32.156, -167.921, -21.557, -11.256]
  MoveL 280 to (-96.48, -14.81, 54) mm, rotated rx -180 ry 0 rz -180 deg; joints [-4.729, -10.958, -32.094, -167.079, -21.635, -12.038]
  MoveL 281 to (-95.43, -20.53, 54) mm, rotated rx -180 ry 0 rz -180 deg; joints [-4.976, -10.878, -32.028, -166.433, -21.702, -12.637]
  MoveL 282 to (-94.18, -25.65, 54) mm, rotated rx 180 ry 0 rz 180 deg; joints [-5.196, -10.789, -31.954, -165.864, -21.766, -13.165]
  MoveL 283 to (-91.95, -32.74, 54) mm, rotated rx 180 ry 0 rz -180 deg; joints [-5.497, -10.638, -31.83, -165.092, -21.861, -13.878]
  MoveL 284 to (-88.96, -40.18, 54) mm, rotated rx -180 ry 0 rz 180 deg; joints [-5.809, -10.444, -31.669, -164.305, -21.97, -14.606]
  MoveL 285 to (-86.2, -45.75, 54) mm, rotated rx 180 ry 0 rz 180 deg; joints [-6.038, -10.27, -31.524, -163.733, -22.057, -15.133]
  MoveL 286 to (-82.9, -51.54, 54) mm, rotated rx -180 ry 0 rz 180 deg; joints [-6.274, -10.066, -31.354, -163.153, -22.152, -15.667]
  MoveL 287 to (-78.03, -58.65, 54) mm, rotated rx -180 ry 0 rz -180 deg; joints [-6.557, -9.772, -31.107, -162.467, -22.275, -16.297]
  MoveL 288 to (-74.07, -63.57, 54) mm, rotated rx -180 ry 0 rz 180 deg; joints [-6.749, -9.538, -30.91, -162.01, -22.364, -16.715]
  MoveL 289 to (-69.24, -68.8, 54) mm, rotated rx 180 ry 0 rz 180 deg; joints [-6.948, -9.256, -30.671, -161.543, -22.463, -17.142]
  MoveL 290 to (-62.87, -74.67, 54) mm, rotated rx -180 ry 0 rz -180 deg; joints [-7.164, -8.891, -30.359, -161.046, -22.579, -17.594]
  MoveL 291 to (-60.57, -76.44, 54) mm, rotated rx -180 ry 0 rz -180 deg; joints [-7.227, -8.761, -30.248, -160.905, -22.615, -17.722]
  Set speed (16.7 mm/s)
  MoveL 292 to (-59.99, -76.68, 54) mm, rotated rx -180 ry 0 rz 180 deg; joints [-7.234, -8.73, -30.221, -160.891, -22.622, -17.735]
  MoveL 293 to (-59.38, -76.6, 54) mm, rotated rx -180 ry 0 rz 180 deg; joints [-7.227, -8.699, -30.195, -160.911, -22.624, -17.716]
  MoveL 294 to (-58.89, -76.22, 54) mm, rotated rx -180 ry 0 rz -180 deg; joints [-7.209, -8.676, -30.175, -160.959, -22.621, -17.67]
  MoveL 295 to (-59.1, -74.54, 54) mm, rotated rx -180 ry 0 rz -180 deg; joints [-7.138, -8.698, -30.194, -161.131, -22.597, -17.512]
  MoveL 296 to (-55.68, -70.05, 54) mm, rotated rx -180 ry 0 rz -180 deg; joints [-6.931, -8.551, -30.067, -161.664, -22.555, -17.018]
  Set speed (5.0 mm/s)
  MoveL 297 to (-55.68, -70.05, 48) mm, rotated rx -180 ry 0 rz 180 deg; joints [-6.931, -8.495, -30.299, -161.878, -22.827, -16.785]
  MoveL 298 to (-57.37, -70.27, 48) mm, rotated rx 180 ry 0 rz 180 deg; joints [-6.949, -8.58, -30.372, -161.825, -22.821, -16.836]
  MoveL 299 to (-57.6, -70.85, 48) mm, rotated rx 180 ry 0 rz 180 deg; joints [-6.974, -8.589, -30.38, -161.761, -22.828, -16.895]
  MoveL 300 to (-57.52, -71.46, 48) mm, rotated rx -180 ry 0 rz -180 deg; joints [-7, -8.581, -30.373, -161.698, -22.836, -16.953]
  MoveL 301 to (-57.14, -71.96, 48) mm, rotated rx -180 ry 0 rz 180 deg; joints [-7.019, -8.558, -30.353, -161.654, -22.845, -16.993]
  Set speed (16.7 mm/s)
  MoveL 302 to (-52.2, -75.73, 48) mm, rotated rx -180 ry 0 rz 180 deg; joints [-7.152, -8.28, -30.113, -161.355, -22.92, -17.264]
  MoveL 303 to (-44.74, -80.37, 48) mm, rotated rx -180 ry 0 rz -180 deg; joints [-7.307, -7.868, -29.755, -161.017, -23.018, -17.568]
  MoveL 304 to (-37.46, -84, 48) mm, rotated rx -180 ry 0 rz -180 deg; joints [-7.42, -7.472, -29.408, -160.782, -23.099, -17.779]
  MoveL 305 to (-36.02, -84.61, 48) mm, rotated rx 180 ry 0 rz 180 deg; joints [-7.437, -7.394, -29.34, -160.747, -23.113, -17.809]
  MoveL 306 to (-28.59, -87.42, 48) mm, rotated rx -180 ry 0 rz -180 deg; joints [-7.513, -6.997, -28.989, -160.598, -23.18, -17.94]
  MoveL 307 to (-22.16, -89.21, 48) mm, rotated rx 180 ry 0 rz -180 deg; joints [-7.552, -6.657, -28.688, -160.534, -23.228, -17.994]
  MoveL 308 to (-16.12, -90.54, 48) mm, rotated rx 180 ry 0 rz 180 deg; joints [-7.574, -6.342, -28.405, -160.507, -23.266, -18.014]
  MoveL 309 to (-8.61, -91.57, 48) mm, rotated rx -180 ry 0 rz -180 deg; joints [-7.575, -5.954, -28.056, -160.534, -23.303, -17.984]
  MoveL 310 to (-1.31, -91.97, 48) mm, rotated rx -180 ry 0 rz -180 deg; joints [-7.552, -5.582, -27.72, -160.617, -23.329, -17.903]
  MoveL 311 to (5.67, -91.8, 48) mm, rotated rx -180 ry 0 rz 180 deg; joints [-7.508, -5.231, -27.399, -160.747, -23.345, -17.78]
  MoveL 312 to (11.76, -91.19, 48) mm, rotated rx 180 ry 0 rz 180 deg; joints [-7.451, -4.927, -27.121, -160.903, -23.351, -17.634]
  MoveL 313 to (18.37, -90.08, 48) mm, rotated rx -180 ry 0 rz -180 deg; joints [-7.372, -4.602, -26.821, -161.111, -23.351, -17.439]
  MoveL 314 to (24.9, -88.54, 48) mm, rotated rx -180 ry 0 rz 180 deg; joints [-7.277, -4.283, -26.525, -161.357, -23.345, -17.21]
  MoveL 315 to (30.95, -86.62, 48) mm, rotated rx -180 ry 0 rz -180 deg; joints [-7.17, -3.992, -26.253, -161.63, -23.332, -16.957]
  MoveL 316 to (37.38, -83.99, 48) mm, rotated rx -180 ry 0 rz -180 deg; joints [-7.034, -3.685, -25.966, -161.972, -23.311, -16.641]
  MoveL 317 to (42.52, -81.53, 48) mm, rotated rx 180 ry 0 rz 180 deg; joints [-6.913, -3.443, -25.738, -162.278, -23.29, -16.359]
  MoveL 318 to (47.96, -78.48, 48) mm, rotated rx -180 ry 0 rz 180 deg; joints [-6.767, -3.189, -25.497, -162.641, -23.262, -16.024]
  MoveL 319 to (48.6, -78.09, 48) mm, rotated rx -180 ry 0 rz 180 deg; joints [-6.749, -3.159, -25.469, -162.686, -23.259, -15.981]
  MoveL 320 to (55.28, -73.51, 48) mm, rotated rx -180 ry 0 rz 180 deg; joints [-6.539, -2.851, -25.177, -163.209, -23.216, -15.5]
  MoveL 321 to (56.61, -72.47, 48) mm, rotated rx -180 ry 0 rz -180 deg; joints [-6.493, -2.79, -25.119, -163.324, -23.207, -15.393]
  MoveL 322 to (62.07, -67.88, 48) mm, rotated rx 180 ry 0 rz 180 deg; joints [-6.289, -2.543, -24.882, -163.829, -23.164, -14.928]
  MoveL 323 to (66.2, -63.79, 48) mm, rotated rx 180 ry 0 rz 180 deg; joints [-6.113, -2.359, -24.705, -164.268, -23.126, -14.523]
  MoveL 324 to (70.26, -59.36, 48) mm, rotated rx 180 ry 0 rz 180 deg; joints [-5.924, -2.179, -24.532, -164.739, -23.086, -14.09]
  MoveL 325 to (74.13, -54.44, 48) mm, rotated rx -180 ry 0 rz 180 deg; joints [-5.719, -2.011, -24.37, -165.252, -23.042, -13.617]
  MoveL 326 to (78.44, -48.03, 48) mm, rotated rx -180 ry 0 rz 180 deg; joints [-5.454, -1.827, -24.192, -165.913, -22.987, -13.008]
  MoveL 327 to (82.11, -41.45, 48) mm, rotated rx 180 ry 0 rz 180 deg; joints [-5.187, -1.675, -24.044, -166.584, -22.932, -12.39]
  MoveL 328 to (85.71, -33.38, 48) mm, rotated rx -180 ry 0 rz -180 deg; joints [-4.864, -1.531, -23.903, -167.398, -22.869, -11.639]
  MoveL 329 to (87.95, -26.82, 48) mm, rotated rx 180 ry 0 rz 180 deg; joints [-4.604, -1.445, -23.82, -168.055, -22.82, -11.034]
  MoveL 330 to (89.39, -21.4, 48) mm, rotated rx -180 ry 0 rz 180 deg; joints [-4.391, -1.395, -23.771, -168.596, -22.781, -10.535]
  MoveL 331 to (90.83, -14.31, 48) mm, rotated rx -180 ry 0 rz 180 deg; joints [-4.114, -1.349, -23.726, -169.301, -22.733, -9.885]
  MoveL 332 to (91.65, -7.73, 48) mm, rotated rx 180 ry 0 rz 180 deg; joints [-3.859, -1.331, -23.709, -169.953, -22.691, -9.284]
  MoveL 333 to (91.96, -1.13, 48) mm, rotated rx -180 ry 0 rz 180 deg; joints [-3.604, -1.337, -23.715, -170.605, -22.651, -8.682]
  MoveL 334 to (91.85, 3.87, 48) mm, rotated rx -180 ry 0 rz -180 deg; joints [-3.412, -1.358, -23.735, -171.099, -22.622, -8.226]
  MoveL 335 to (91.35, 10.46, 48) mm, rotated rx -180 ry 0 rz 180 deg; joints [-3.159, -1.402, -23.778, -171.75, -22.586, -7.625]
  MoveL 336 to (90.17, 17.98, 48) mm, rotated rx 180 ry 0 rz 180 deg; joints [-2.872, -1.481, -23.855, -172.492, -22.548, -6.94]
  MoveL 337 to (88.12, 26.32, 48) mm, rotated rx 180 ry 0 rz 180 deg; joints [-2.554, -1.603, -23.974, -173.317, -22.509, -6.178]
  MoveL 338 to (85.9, 32.86, 48) mm, rotated rx 180 ry 0 rz 180 deg; joints [-2.304, -1.729, -24.096, -173.965, -22.48, -5.58]
  MoveL 339 to (85.32, 34.32, 48) mm, rotated rx 180 ry 0 rz 180 deg; joints [-2.248, -1.76, -24.127, -174.109, -22.474, -5.446]
  MoveL 340 to (82.39, 40.87, 48) mm, rotated rx -180 ry 0 rz -180 deg; joints [-1.999, -1.919, -24.281, -174.759, -22.446, -4.846]
  MoveL 341 to (82.22, 41.22, 48) mm, rotated rx -180 ry 0 rz 180 deg; joints [-1.985, -1.928, -24.29, -174.794, -22.445, -4.814]
  MoveL 342 to (77.98, 48.77, 48) mm, rotated rx 180 ry 0 rz 180 deg; joints [-1.697, -2.153, -24.507, -175.546, -22.415, -4.118]
  MoveL 343 to (73.26, 55.61, 48) mm, rotated rx 180 ry 0 rz 180 deg; joints [-1.435, -2.4, -24.744, -176.23, -22.388, -3.486]
  MoveL 344 to (68.95, 60.83, 48) mm, rotated rx 180 ry 0 rz 180 deg; joints [-1.234, -2.623, -24.959, -176.755, -22.368, -3.001]
  MoveL 345 to (64.76, 65.31, 48) mm, rotated rx -180 ry 0 rz 180 deg; joints [-1.062, -2.838, -25.164, -177.207, -22.35, -2.583]
  MoveL 346 to (59.26, 70.34, 48) mm, rotated rx -180 ry 0 rz 180 deg; joints [-0.867, -3.119, -25.432, -177.717, -22.328, -2.112]
  MoveL 347 to (52.28, 75.67, 48) mm, rotated rx 180 ry 0 rz 180 deg; joints [-0.66, -3.475, -25.768, -178.262, -22.302, -1.608]
  MoveL 348 to (44.7, 80.38, 48) mm, rotated rx 180 ry 0 rz 180 deg; joints [-0.475, -3.861, -26.131, -178.746, -22.275, -1.16]
  MoveL 349 to (37.42, 84.02, 48) mm, rotated rx 180 ry 0 rz 180 deg; joints [-0.332, -4.231, -26.476, -179.124, -22.248, -0.811]
  MoveL 350 to (35.99, 84.62, 48) mm, rotated rx -180 ry 0 rz -180 deg; joints [-0.308, -4.303, -26.544, -179.186, -22.243, -0.753]
  MoveL 351 to (28.55, 87.43, 48) mm, rotated rx 180 ry 0 rz 180 deg; joints [-0.196, -4.681, -26.894, -179.481, -22.214, -0.48]
  MoveL 352 to (22.12, 89.22, 48) mm, rotated rx -180 ry 0 rz 180 deg; joints [-0.124, -5.008, -27.195, -179.671, -22.187, -0.305]
  MoveL 353 to (16.08, 90.55, 48) mm, rotated rx 180 ry 0 rz 180 deg; joints [-0.071, -5.316, -27.477, -179.812, -22.161, -0.174]
  MoveL 354 to (9.71, 91.46, 48) mm, rotated rx 180 ry 0 rz 180 deg; joints [-0.034, -5.64, -27.773, -179.91, -22.132, -0.083]
  MoveL 355 to (1.28, 91.97, 48) mm, rotated rx 180 ry 0 rz 180 deg; joints [-0.013, -6.071, -28.162, -179.965, -22.091, -0.033]
  MoveL 356 to (-5.71, 91.8, 48) mm, rotated rx -180 ry 0 rz -180 deg; joints [-0.02, -6.428, -28.483, -179.946, -22.055, -0.05]
  MoveL 357 to (-11.8, 91.19, 48) mm, rotated rx -180 ry 0 rz 180 deg; joints [-0.046, -6.74, -28.762, -179.878, -22.021, -0.113]
  MoveL 358 to (-18.41, 90.08, 48) mm, rotated rx -180 ry 0 rz 180 deg; joints [-0.092, -7.079, -29.063, -179.753, -21.983, -0.229]
  MoveL 359 to (-25.03, 88.51, 48) mm, rotated rx -180 ry 0 rz -180 deg; joints [-0.159, -7.42, -29.363, -179.575, -21.943, -0.394]
  MoveL 360 to (-30.89, 86.64, 48) mm, rotated rx -180 ry 0 rz -180 deg; joints [-0.238, -7.721, -29.627, -179.362, -21.907, -0.592]
  MoveL 361 to (-37.32, 84.01, 48) mm, rotated rx 180 ry 0 rz 180 deg; joints [-0.35, -8.053, -29.916, -179.059, -21.866, -0.873]
  MoveL 362 to (-42.55, 81.51, 48) mm, rotated rx -180 ry 0 rz 180 deg; joints [-0.458, -8.322, -30.15, -178.768, -21.832, -1.143]
  MoveL 363 to (-47.99, 78.46, 48) mm, rotated rx -180 ry 0 rz 180 deg; joints [-0.59, -8.602, -30.391, -178.411, -21.796, -1.475]
  MoveL 364 to (-48.63, 78.07, 48) mm, rotated rx 180 ry 0 rz 180 deg; joints [-0.607, -8.635, -30.419, -178.365, -21.792, -1.518]
  MoveL 365 to (-55.31, 73.49, 48) mm, rotated rx 180 ry 0 rz 180 deg; joints [-0.806, -8.979, -30.714, -177.823, -21.749, -2.022]
  MoveL 366 to (-56.64, 72.45, 48) mm, rotated rx -180 ry 0 rz 180 deg; joints [-0.852, -9.047, -30.772, -177.7, -21.741, -2.137]
  MoveL 367 to (-62.1, 67.85, 48) mm, rotated rx 180 ry 0 rz 180 deg; joints [-1.054, -9.327, -31.01, -177.15, -21.708, -2.648]
  MoveL 368 to (-66.23, 63.76, 48) mm, rotated rx -180 ry 0 rz -180 deg; joints [-1.234, -9.537, -31.188, -176.66, -21.684, -3.104]
  MoveL 369 to (-70.29, 59.32, 48) mm, rotated rx 180 ry 0 rz 180 deg; joints [-1.43, -9.744, -31.362, -176.124, -21.664, -3.603]
  MoveL 370 to (-74.08, 54.52, 48) mm, rotated rx -180 ry 0 rz -180 deg; joints [-1.643, -9.935, -31.523, -175.543, -21.648, -4.144]
  MoveL 371 to (-78.47, 47.98, 48) mm, rotated rx -180 ry 0 rz 180 deg; joints [-1.933, -10.153, -31.706, -174.75, -21.635, -4.882]
  MoveL 372 to (-82.06, 41.54, 48) mm, rotated rx 180 ry 0 rz 180 deg; joints [-2.22, -10.329, -31.852, -173.969, -21.632, -5.609]
  MoveL 373 to (-85.66, 33.5, 48) mm, rotated rx -180 ry 0 rz -180 deg; joints [-2.579, -10.499, -31.994, -172.993, -21.642, -6.518]
  MoveL 374 to (-87.91, 26.95, 48) mm, rotated rx -180 ry 0 rz -180 deg; joints [-2.87, -10.601, -32.078, -172.203, -21.659, -7.253]
  MoveL 375 to (-88.49, 25.1, 48) mm, rotated rx -180 ry 0 rz 180 deg; joints [-2.952, -10.626, -32.099, -171.98, -21.666, -7.46]
  MoveL 376 to (-90.47, 16.57, 48) mm, rotated rx -180 ry 0 rz 180 deg; joints [-3.332, -10.705, -32.165, -170.958, -21.704, -8.41]
  MoveL 377 to (-90.85, 14.2, 48) mm, rotated rx -180 ry 0 rz -180 deg; joints [-3.437, -10.718, -32.175, -170.677, -21.718, -8.671]
  MoveL 378 to (-91.63, 7.94, 48) mm, rotated rx 180 ry 0 rz 180 deg; joints [-3.714, -10.738, -32.192, -169.937, -21.758, -9.359]
  MoveL 379 to (-91.91, 2.88, 48) mm, rotated rx -180 ry 0 rz 180 deg; joints [-3.937, -10.735, -32.189, -169.344, -21.796, -9.91]
  MoveL 380 to (-91.88, -2.84, 48) mm, rotated rx -180 ry 0 rz 180 deg; joints [-4.187, -10.712, -32.17, -168.682, -21.844, -10.524]
  MoveL 381 to (-91.5, -9.31, 48) mm, rotated rx -180 ry 0 rz -180 deg; joints [-4.47, -10.667, -32.133, -167.942, -21.905, -11.211]
  MoveL 382 to (-90.64, -15.62, 48) mm, rotated rx 180 ry 0 rz -180 deg; joints [-4.743, -10.595, -32.073, -167.232, -21.972, -11.868]
  MoveL 383 to (-89.73, -19.97, 48) mm, rotated rx -180 ry 0 rz -180 deg; joints [-4.93, -10.529, -32.018, -166.75, -22.022, -12.314]
  MoveL 384 to (-87.98, -26.75, 48) mm, rotated rx 180 ry 0 rz -180 deg; joints [-5.219, -10.406, -31.916, -166.012, -22.105, -12.996]
  MoveL 385 to (-85.97, -32.64, 48) mm, rotated rx 180 ry 0 rz 180 deg; joints [-5.467, -10.273, -31.806, -165.384, -22.184, -13.576]
  MoveL 386 to (-85.38, -34.19, 48) mm, rotated rx 180 ry 0 rz 180 deg; joints [-5.532, -10.234, -31.773, -165.221, -22.206, -13.726]
  MoveL 387 to (-82.28, -41.12, 48) mm, rotated rx -180 ry 0 rz 180 deg; joints [-5.82, -10.037, -31.608, -164.505, -22.307, -14.385]
  MoveL 388 to (-77.89, -48.91, 48) mm, rotated rx 180 ry 0 rz 180 deg; joints [-6.137, -9.767, -31.382, -163.729, -22.429, -15.098]
  MoveL 389 to (-73.31, -55.54, 48) mm, rotated rx -180 ry 0 rz 180 deg; joints [-6.4, -9.492, -31.15, -163.094, -22.54, -15.68]
  MoveL 390 to (-72.91, -56.07, 48) mm, rotated rx 180 ry 0 rz 180 deg; joints [-6.421, -9.468, -31.13, -163.044, -22.55, -15.727]
  MoveL 391 to (-68.99, -60.78, 48) mm, rotated rx -180 ry 0 rz 180 deg; joints [-6.604, -9.237, -30.934, -162.612, -22.633, -16.121]
  MoveL 392 to (-64.81, -65.27, 48) mm, rotated rx -180 ry 0 rz 180 deg; joints [-6.774, -8.995, -30.727, -162.213, -22.715, -16.485]
  MoveL 393 to (-59.3, -70.31, 48) mm, rotated rx 180 ry 0 rz 180 deg; joints [-6.96, -8.68, -30.458, -161.786, -22.812, -16.873]
  MoveL 394 to (-57.14, -71.96, 48) mm, rotated rx -180 ry 0 rz 180 deg; joints [-7.019, -8.558, -30.353, -161.654, -22.845, -16.993]
  Set speed (16.7 mm/s)
  MoveL 395 to (-56.57, -72.19, 48) mm, rotated rx 180 ry 0 rz 180 deg; joints [-7.026, -8.527, -30.326, -161.64, -22.851, -17.005]
  MoveL 396 to (-55.95, -72.11, 48) mm, rotated rx -180 ry 0 rz 180 deg; joints [-7.019, -8.496, -30.3, -161.66, -22.853, -16.987]
  MoveL 397 to (-55.46, -71.73, 48) mm, rotated rx -180 ry 0 rz -180 deg; joints [-7.001, -8.473, -30.28, -161.708, -22.851, -16.942]
  MoveL 398 to (-55.69, -70.04, 48) mm, rotated rx -180 ry 0 rz 180 deg; joints [-6.931, -8.495, -30.299, -161.878, -22.827, -16.785]
  MoveL 399 to (-51.73, -64.96, 48) mm, rotated rx 180 ry 0 rz -180 deg; joints [-6.696, -8.324, -30.151, -162.476, -22.783, -16.231]
  Set speed (5.0 mm/s)
  MoveL 400 to (-51.73, -64.96, 42) mm, rotated rx -180 ry 0 rz -180 deg; joints [-6.696, -8.266, -30.381, -162.68, -23.057, -16.01]
  MoveL 401 to (-53.42, -65.17, 42) mm, rotated rx -180 ry 0 rz -180 deg; joints [-6.713, -8.352, -30.455, -162.629, -23.051, -16.058]
  MoveL 402 to (-53.66, -65.75, 42) mm, rotated rx -180 ry 0 rz 180 deg; joints [-6.739, -8.361, -30.462, -162.566, -23.057, -16.117]
  MoveL 403 to (-53.58, -66.36, 42) mm, rotated rx 180 ry 0 rz 180 deg; joints [-6.764, -8.353, -30.456, -162.504, -23.065, -16.174]
  MoveL 404 to (-53.2, -66.86, 42) mm, rotated rx -180 ry 0 rz -180 deg; joints [-6.783, -8.33, -30.436, -162.459, -23.073, -16.214]
  Set speed (16.7 mm/s)
  MoveL 405 to (-48.61, -70.41, 42) mm, rotated rx 180 ry 0 rz 180 deg; joints [-6.91, -8.072, -30.213, -162.175, -23.142, -16.472]
  MoveL 406 to (-44.8, -72.87, 42) mm, rotated rx -180 ry 0 rz -180 deg; joints [-6.994, -7.862, -30.029, -161.99, -23.192, -16.639]
  MoveL 407 to (-42.05, -74.51, 42) mm, rotated rx -180 ry 0 rz -180 deg; joints [-7.048, -7.711, -29.898, -161.871, -23.225, -16.745]
  MoveL 408 to (-36.66, -77.31, 42) mm, rotated rx -180 ry 0 rz 180 deg; joints [-7.137, -7.417, -29.64, -161.683, -23.285, -16.914]
  MoveL 409 to (-29.93, -80.15, 42) mm, rotated rx 180 ry 0 rz 180 deg; joints [-7.22, -7.055, -29.321, -161.513, -23.35, -17.064]
  MoveL 410 to (-23.97, -82.13, 42) mm, rotated rx -180 ry 0 rz 180 deg; joints [-7.27, -6.739, -29.04, -161.418, -23.399, -17.147]
  MoveL 411 to (-17.15, -83.82, 42) mm, rotated rx -180 ry 0 rz -180 deg; joints [-7.304, -6.381, -28.72, -161.365, -23.445, -17.191]
  MoveL 412 to (-9.82, -84.99, 42) mm, rotated rx -180 ry 0 rz 180 deg; joints [-7.313, -6.001, -28.379, -161.371, -23.484, -17.181]
  MoveL 413 to (-3.83, -85.47, 42) mm, rotated rx -180 ry 0 rz -180 deg; joints [-7.302, -5.695, -28.102, -161.42, -23.508, -17.132]
  MoveL 414 to (3.69, -85.48, 42) mm, rotated rx -180 ry 0 rz -180 deg; joints [-7.263, -5.314, -27.755, -161.538, -23.529, -17.019]
  MoveL 415 to (11.2, -84.82, 42) mm, rotated rx -180 ry 0 rz 180 deg; joints [-7.198, -4.939, -27.412, -161.716, -23.54, -16.852]
  MoveL 416 to (18.29, -83.58, 42) mm, rotated rx 180 ry 0 rz 180 deg; joints [-7.113, -4.589, -27.089, -161.941, -23.541, -16.643]
  MoveL 417 to (25.56, -81.65, 42) mm, rotated rx -180 ry 0 rz -180 deg; joints [-6.999, -4.235, -26.761, -162.23, -23.534, -16.374]
  MoveL 418 to (31.67, -79.48, 42) mm, rotated rx -180 ry 0 rz 180 deg; joints [-6.884, -3.941, -26.486, -162.522, -23.52, -16.104]
  MoveL 419 to (37.31, -76.99, 42) mm, rotated rx -180 ry 0 rz -180 deg; joints [-6.758, -3.673, -26.235, -162.836, -23.501, -15.815]
  MoveL 420 to (43.88, -73.45, 42) mm, rotated rx -180 ry 0 rz -180 deg; joints [-6.588, -3.364, -25.944, -163.259, -23.473, -15.424]
  MoveL 421 to (49.69, -69.65, 42) mm, rotated rx -180 ry 0 rz 180 deg; joints [-6.413, -3.095, -25.688, -163.694, -23.44, -15.024]
  MoveL 422 to (54.94, -65.59, 42) mm, rotated rx 180 ry 0 rz -180 deg; joints [-6.231, -2.854, -25.46, -164.144, -23.405, -14.61]
  MoveL 423 to (60.24, -60.71, 42) mm, rotated rx 180 ry 0 rz 180 deg; joints [-6.018, -2.615, -25.231, -164.67, -23.362, -14.125]
  MoveL 424 to (65.67, -54.84, 42) mm, rotated rx 180 ry 0 rz 180 deg; joints [-5.767, -2.374, -25, -165.291, -23.312, -13.555]
  MoveL 425 to (70.17, -48.95, 42) mm, rotated rx 180 ry 0 rz 180 deg; joints [-5.521, -2.178, -24.811, -165.902, -23.262, -12.993]
  MoveL 426 to (72.56, -45.34, 42) mm, rotated rx -180 ry 0 rz 180 deg; joints [-5.372, -2.076, -24.712, -166.272, -23.233, -12.652]
  MoveL 427 to (75.64, -39.99, 42) mm, rotated rx -180 ry 0 rz 180 deg; joints [-5.153, -1.946, -24.587, -166.815, -23.19, -12.152]
  MoveL 428 to (77.2, -36.88, 42) mm, rotated rx 180 ry 0 rz 180 deg; joints [-5.027, -1.882, -24.525, -167.129, -23.166, -11.864]
  MoveL 429 to (79.63, -31.29, 42) mm, rotated rx -180 ry 0 rz 180 deg; joints [-4.803, -1.785, -24.431, -167.69, -23.123, -11.348]
  MoveL 430 to (81.31, -26.62, 42) mm, rotated rx 180 ry 0 rz 180 deg; joints [-4.617, -1.72, -24.368, -168.155, -23.089, -10.92]
  MoveL 431 to (83.39, -19.15, 42) mm, rotated rx 180 ry 0 rz 180 deg; joints [-4.322, -1.645, -24.295, -168.897, -23.037, -10.237]
  MoveL 432 to (84.88, -10.72, 42) mm, rotated rx -180 ry 0 rz 180 deg; joints [-3.992, -1.601, -24.252, -169.729, -22.982, -9.471]
  MoveL 433 to (85.5, -3.04, 42) mm, rotated rx 180 ry 0 rz 180 deg; joints [-3.694, -1.596, -24.247, -170.484, -22.935, -8.776]
  MoveL 434 to (85.44, 4.45, 42) mm, rotated rx -180 ry 0 rz -180 deg; joints [-3.404, -1.622, -24.273, -171.219, -22.892, -8.099]
  MoveL 435 to (84.81, 11.19, 42) mm, rotated rx 180 ry 0 rz 180 deg; joints [-3.145, -1.673, -24.322, -171.88, -22.855, -7.49]
  MoveL 436 to (83.78, 17.33, 42) mm, rotated rx 180 ry 0 rz 180 deg; joints [-2.909, -1.741, -24.388, -172.481, -22.824, -6.936]
  MoveL 437 to (81.66, 25.53, 42) mm, rotated rx 180 ry 0 rz 180 deg; joints [-2.595, -1.867, -24.51, -173.285, -22.784, -6.195]
  MoveL 438 to (79.72, 31.05, 42) mm, rotated rx 180 ry 0 rz 180 deg; joints [-2.384, -1.976, -24.616, -173.827, -22.759, -5.696]
  MoveL 439 to (76.91, 37.48, 42) mm, rotated rx -180 ry 0 rz 180 deg; joints [-2.138, -2.13, -24.765, -174.458, -22.73, -5.114]
  MoveL 440 to (73.66, 43.52, 42) mm, rotated rx -180 ry 0 rz -180 deg; joints [-1.907, -2.304, -24.932, -175.054, -22.705, -4.564]
  MoveL 441 to (69.28, 50.21, 42) mm, rotated rx -180 ry 0 rz -180 deg; joints [-1.651, -2.534, -25.154, -175.715, -22.676, -3.955]
  MoveL 442 to (65.29, 55.29, 42) mm, rotated rx -180 ry 0 rz -180 deg; joints [-1.455, -2.742, -25.352, -176.22, -22.655, -3.489]
  MoveL 443 to (60.71, 60.28, 42) mm, rotated rx -180 ry 0 rz 180 deg; joints [-1.263, -2.979, -25.578, -176.717, -22.633, -3.031]
  MoveL 444 to (55.8, 64.86, 42) mm, rotated rx -180 ry 0 rz -180 deg; joints [-1.086, -3.231, -25.818, -177.174, -22.611, -2.609]
  MoveL 445 to (49.38, 69.86, 42) mm, rotated rx -180 ry 0 rz -180 deg; joints [-0.892, -3.559, -26.128, -177.677, -22.585, -2.145]
  MoveL 446 to (44.75, 72.91, 42) mm, rotated rx 180 ry 0 rz 180 deg; joints [-0.773, -3.795, -26.35, -177.984, -22.567, -1.861]
  MoveL 447 to (40.32, 75.46, 42) mm, rotated rx -180 ry 0 rz -180 deg; joints [-0.674, -4.022, -26.561, -178.243, -22.549, -1.623]
  MoveL 448 to (34.07, 78.48, 42) mm, rotated rx 180 ry 0 rz 180 deg; joints [-0.555, -4.34, -26.858, -178.551, -22.524, -1.339]
  MoveL 449 to (26.74, 81.27, 42) mm, rotated rx 180 ry 0 rz 180 deg; joints [-0.445, -4.713, -27.204, -178.836, -22.495, -1.075]
  MoveL 450 to (19.02, 83.42, 42) mm, rotated rx -180 ry 0 rz 180 deg; joints [-0.361, -5.106, -27.565, -179.056, -22.462, -0.872]
  MoveL 451 to (11.45, 84.79, 42) mm, rotated rx -180 ry 0 rz 180 deg; joints [-0.307, -5.493, -27.918, -179.196, -22.427, -0.743]
  MoveL 452 to (3.9, 85.47, 42) mm, rotated rx -180 ry 0 rz 180 deg; joints [-0.28, -5.878, -28.268, -179.264, -22.391, -0.68]
  MoveL 453 to (-3.73, 85.48, 42) mm, rotated rx -180 ry 0 rz 180 deg; joints [-0.281, -6.268, -28.619, -179.26, -22.353, -0.685]
  MoveL 454 to (-11.23, 84.82, 42) mm, rotated rx 180 ry 0 rz 180 deg; joints [-0.31, -6.653, -28.963, -179.182, -22.313, -0.756]
  MoveL 455 to (-18.23, 83.59, 42) mm, rotated rx 180 ry 0 rz 180 deg; joints [-0.363, -7.011, -29.282, -179.042, -22.273, -0.886]
  MoveL 456 to (-25.59, 81.64, 42) mm, rotated rx -180 ry 0 rz 180 deg; joints [-0.447, -7.39, -29.616, -178.818, -22.23, -1.094]
  MoveL 457 to (-31.7, 79.47, 42) mm, rotated rx 180 ry 0 rz 180 deg; joints [-0.54, -7.703, -29.891, -178.569, -22.194, -1.325]
  MoveL 458 to (-37.34, 76.98, 42) mm, rotated rx 180 ry 0 rz 180 deg; joints [-0.648, -7.993, -30.144, -178.281, -22.16, -1.592]
  MoveL 459 to (-43.91, 73.43, 42) mm, rotated rx -180 ry 0 rz -180 deg; joints [-0.802, -8.331, -30.436, -177.869, -22.12, -1.974]
  MoveL 460 to (-49.72, 69.63, 42) mm, rotated rx 180 ry 0 rz 180 deg; joints [-0.968, -8.628, -30.693, -177.425, -22.085, -2.386]
  MoveL 461 to (-54.88, 65.64, 42) mm, rotated rx 180 ry 0 rz 180 deg; joints [-1.143, -8.892, -30.92, -176.956, -22.055, -2.822]
  MoveL 462 to (-60.27, 60.68, 42) mm, rotated rx -180 ry 0 rz 180 deg; joints [-1.361, -9.167, -31.154, -176.37, -22.027, -3.366]
  MoveL 463 to (-65.69, 54.81, 42) mm, rotated rx 180 ry 0 rz 180 deg; joints [-1.62, -9.441, -31.387, -175.673, -22.002, -4.013]
  MoveL 464 to (-70.12, 49.02, 42) mm, rotated rx -180 ry 0 rz 180 deg; joints [-1.876, -9.663, -31.574, -174.984, -21.987, -4.653]
  MoveL 465 to (-72.58, 45.3, 42) mm, rotated rx -180 ry 0 rz -180 deg; joints [-2.041, -9.785, -31.676, -174.54, -21.982, -5.066]
  MoveL 466 to (-75.59, 40.08, 42) mm, rotated rx -180 ry 0 rz 180 deg; joints [-2.273, -9.931, -31.799, -173.918, -21.98, -5.643]
  MoveL 467 to (-77.15, 36.98, 42) mm, rotated rx -180 ry 0 rz -180 deg; joints [-2.41, -10.006, -31.862, -173.549, -21.982, -5.986]
  MoveL 468 to (-79.65, 31.24, 42) mm, rotated rx -180 ry 0 rz 180 deg; joints [-2.665, -10.123, -31.96, -172.866, -21.991, -6.62]
  MoveL 469 to (-81.27, 26.75, 42) mm, rotated rx -180 ry 0 rz -180 deg; joints [-2.864, -10.196, -32.021, -172.335, -22.003, -7.112]
  MoveL 470 to (-83.35, 19.31, 42) mm, rotated rx 180 ry 0 rz 180 deg; joints [-3.194, -10.285, -32.095, -171.458, -22.032, -7.926]
  MoveL 471 to (-84.86, 10.93, 42) mm, rotated rx 180 ry 0 rz 180 deg; joints [-3.564, -10.338, -32.139, -170.48, -22.077, -8.834]
  MoveL 472 to (-85.49, 3.34, 42) mm, rotated rx 180 ry 0 rz 180 deg; joints [-3.897, -10.345, -32.145, -169.605, -22.129, -9.644]
  MoveL 473 to (-85.42, -4.74, 42) mm, rotated rx 180 ry 0 rz 180 deg; joints [-4.25, -10.311, -32.117, -168.687, -22.196, -10.494]
  MoveL 474 to (-84.72, -11.87, 42) mm, rotated rx 180 ry 0 rz 180 deg; joints [-4.559, -10.246, -32.063, -167.891, -22.265, -11.23]
  MoveL 475 to (-83.37, -19.19, 42) mm, rotated rx 180 ry 0 rz 180 deg; joints [-4.872, -10.144, -31.978, -167.09, -22.345, -11.97]
  MoveL 476 to (-81.74, -25.26, 42) mm, rotated rx -180 ry 0 rz -180 deg; joints [-5.13, -10.032, -31.884, -166.44, -22.417, -12.569]
  MoveL 477 to (-79.79, -30.88, 42) mm, rotated rx 180 ry 0 rz 180 deg; joints [-5.366, -9.903, -31.776, -165.85, -22.49, -13.112]
  MoveL 478 to (-76.81, -37.7, 42) mm, rotated rx -180 ry 0 rz 180 deg; joints [-5.648, -9.714, -31.617, -165.152, -22.585, -13.755]
  MoveL 479 to (-73.71, -43.43, 42) mm, rotated rx -180 ry 0 rz 180 deg; joints [-5.882, -9.523, -31.456, -164.58, -22.67, -14.279]
  MoveL 480 to (-69.33, -50.14, 42) mm, rotated rx -180 ry 0 rz 180 deg; joints [-6.15, -9.26, -31.232, -163.935, -22.776, -14.87]
  MoveL 481 to (-65.2, -55.39, 42) mm, rotated rx -180 ry 0 rz 180 deg; joints [-6.355, -9.017, -31.026, -163.448, -22.864, -15.315]
  MoveL 482 to (-60.75, -60.24, 42) mm, rotated rx 180 ry 0 rz 180 deg; joints [-6.54, -8.759, -30.805, -163.015, -22.949, -15.709]
  MoveL 483 to (-55.84, -64.82, 42) mm, rotated rx -180 ry 0 rz -180 deg; joints [-6.71, -8.478, -30.564, -162.624, -23.034, -16.065]
  MoveL 484 to (-53.2, -66.86, 42) mm, rotated rx -180 ry 0 rz -180 deg; joints [-6.783, -8.33, -30.436, -162.459, -23.073, -16.214]
  Set speed (16.7 mm/s)
  MoveL 485 to (-52.63, -67.1, 42) mm, rotated rx -180 ry 0 rz -180 deg; joints [-6.791, -8.299, -30.409, -162.444, -23.079, -16.227]
  MoveL 486 to (-52.02, -67.02, 42) mm, rotated rx 180 ry 0 rz -180 deg; joints [-6.784, -8.268, -30.382, -162.463, -23.081, -16.21]
  MoveL 487 to (-51.52, -66.64, 42) mm, rotated rx 180 ry 0 rz -180 deg; joints [-6.766, -8.245, -30.363, -162.51, -23.079, -16.166]
  MoveL 488 to (-51.74, -64.95, 42) mm, rotated rx -180 ry 0 rz -180 deg; joints [-6.696, -8.267, -30.381, -162.68, -23.057, -16.01]
  MoveL 489 to (-46.77, -59.56, 42) mm, rotated rx -180 ry 0 rz 180 deg; joints [-6.444, -8.043, -30.187, -163.319, -23.017, -15.418]
  Set speed (5.0 mm/s)
  MoveL 490 to (-46.77, -59.56, 36) mm, rotated rx -180 ry 0 rz -180 deg; joints [-6.444, -7.984, -30.416, -163.511, -23.293, -15.21]
  MoveL 491 to (-48.47, -59.66, 36) mm, rotated rx -180 ry 0 rz 180 deg; joints [-6.457, -8.071, -30.491, -163.473, -23.285, -15.246]
  MoveL 492 to (-48.74, -60.22, 36) mm, rotated rx 180 ry 0 rz 180 deg; joints [-6.481, -8.082, -30.501, -163.412, -23.29, -15.303]
  MoveL 493 to (-48.7, -60.84, 36) mm, rotated rx 180 ry 0 rz 180 deg; joints [-6.507, -8.076, -30.496, -163.349, -23.298, -15.36]
  MoveL 494 to (-48.36, -61.36, 36) mm, rotated rx -180 ry 0 rz -180 deg; joints [-6.528, -8.056, -30.478, -163.302, -23.306, -15.403]
  Set speed (16.7 mm/s)
  MoveL 495 to (-47.98, -61.7, 36) mm, rotated rx -180 ry 0 rz 180 deg; joints [-6.54, -8.034, -30.459, -163.273, -23.312, -15.429]
  MoveL 496 to (-42.49, -65.55, 36) mm, rotated rx 180 ry 0 rz 180 deg; joints [-6.675, -7.729, -30.193, -162.971, -23.386, -15.701]
  MoveL 497 to (-40.06, -67.1, 36) mm, rotated rx -180 ry 0 rz 180 deg; joints [-6.728, -7.596, -30.077, -162.854, -23.416, -15.807]
  MoveL 498 to (-33.19, -70.76, 36) mm, rotated rx 180 ry 0 rz 180 deg; joints [-6.846, -7.221, -29.748, -162.599, -23.492, -16.036]
  MoveL 499 to (-26.91, -73.37, 36) mm, rotated rx -180 ry 0 rz 180 deg; joints [-6.924, -6.885, -29.45, -162.44, -23.55, -16.177]
  MoveL 500 to (-20.54, -75.37, 36) mm, rotated rx -180 ry 0 rz -180 deg; joints [-6.974, -6.548, -29.15, -162.345, -23.599, -16.26]
  MoveL 501 to (-14.27, -76.84, 36) mm, rotated rx -180 ry 0 rz 180 deg; joints [-7.003, -6.22, -28.856, -162.3, -23.64, -16.297]
  MoveL 502 to (-13.75, -76.93, 36) mm, rotated rx -180 ry 0 rz -180 deg; joints [-7.004, -6.192, -28.831, -162.298, -23.643, -16.298]
  MoveL 503 to (-5.11, -77.99, 36) mm, rotated rx -180 ry 0 rz -180 deg; joints [-7.004, -5.747, -28.43, -162.329, -23.684, -16.264]
  MoveL 504 to (-4.8, -78.01, 36) mm, rotated rx -180 ry 0 rz -180 deg; joints [-7.003, -5.732, -28.415, -162.332, -23.685, -16.262]
  MoveL 505 to (2.84, -78.1, 36) mm, rotated rx -180 ry 0 rz 180 deg; joints [-6.969, -5.344, -28.063, -162.438, -23.709, -16.161]
  MoveL 506 to (8.96, -77.63, 36) mm, rotated rx -180 ry 0 rz 180 deg; joints [-6.919, -5.037, -27.782, -162.573, -23.72, -16.033]
  MoveL 507 to (16.36, -76.42, 36) mm, rotated rx -180 ry 0 rz 180 deg; joints [-6.835, -4.671, -27.445, -162.795, -23.725, -15.827]
  MoveL 508 to (24.3, -74.27, 36) mm, rotated rx -180 ry 0 rz 180 deg; joints [-6.711, -4.283, -27.086, -163.11, -23.719, -15.535]
  MoveL 509 to (32.46, -71.09, 36) mm, rotated rx -180 ry 0 rz 180 deg; joints [-6.547, -3.891, -26.72, -163.521, -23.7, -15.155]
  MoveL 510 to (40.98, -66.55, 36) mm, rotated rx 180 ry 0 rz 180 deg; joints [-6.329, -3.489, -26.342, -164.062, -23.668, -14.658]
  MoveL 511 to (44.33, -64.31, 36) mm, rotated rx 180 ry 0 rz 180 deg; joints [-6.226, -3.333, -26.195, -164.316, -23.65, -14.424]
  MoveL 512 to (50.31, -59.8, 36) mm, rotated rx -180 ry 0 rz -180 deg; joints [-6.023, -3.057, -25.933, -164.815, -23.614, -13.965]
  MoveL 513 to (55.95, -54.56, 36) mm, rotated rx 180 ry 0 rz 180 deg; joints [-5.794, -2.802, -25.69, -165.377, -23.572, -13.449]
  MoveL 514 to (56.38, -54.12, 36) mm, rotated rx 180 ry 0 rz 180 deg; joints [-5.776, -2.782, -25.671, -165.423, -23.568, -13.407]
  MoveL 515 to (60.65, -49.17, 36) mm, rotated rx -180 ry 0 rz 180 deg; joints [-5.565, -2.593, -25.49, -165.941, -23.528, -12.931]
  MoveL 516 to (62.32, -47.17, 36) mm, rotated rx -180 ry 0 rz -180 deg; joints [-5.481, -2.519, -25.42, -166.149, -23.513, -12.74]
  MoveL 517 to (67.49, -39.4, 36) mm, rotated rx -180 ry 0 rz -180 deg; joints [-5.159, -2.296, -25.205, -166.943, -23.452, -12.011]
  MoveL 518 to (67.8, -38.87, 36) mm, rotated rx 180 ry 0 rz -180 deg; joints [-5.137, -2.283, -25.193, -166.996, -23.448, -11.962]
  MoveL 519 to (71.95, -30.49, 36) mm, rotated rx -180 ry 0 rz 180 deg; joints [-4.797, -2.112, -25.028, -167.837, -23.386, -11.19]
  MoveL 520 to (72.38, -29.49, 36) mm, rotated rx 180 ry 0 rz 180 deg; joints [-4.756, -2.095, -25.011, -167.938, -23.379, -11.097]
  MoveL 521 to (74.52, -23.42, 36) mm, rotated rx -180 ry 0 rz -180 deg; joints [-4.514, -2.013, -24.932, -168.54, -23.336, -10.545]
  MoveL 522 to (76.17, -17.51, 36) mm, rotated rx -180 ry 0 rz -180 deg; joints [-4.279, -1.952, -24.874, -169.124, -23.296, -10.008]
  MoveL 523 to (77.24, -11.75, 36) mm, rotated rx 180 ry 0 rz 180 deg; joints [-4.053, -1.92, -24.842, -169.69, -23.259, -9.488]
  MoveL 524 to (78.03, -4.42, 36) mm, rotated rx 180 ry 0 rz 180 deg; joints [-3.766, -1.906, -24.828, -170.407, -23.213, -8.829]
  MoveL 525 to (78.15, -0.13, 36) mm, rotated rx -180 ry 0 rz -180 deg; joints [-3.599, -1.913, -24.836, -170.826, -23.188, -8.444]
  MoveL 526 to (77.95, 5.36, 36) mm, rotated rx -180 ry 0 rz 180 deg; joints [-3.386, -1.94, -24.861, -171.362, -23.157, -7.952]
  MoveL 527 to (77.17, 12.37, 36) mm, rotated rx -180 ry 0 rz -180 deg; joints [-3.116, -1.999, -24.919, -172.043, -23.119, -7.325]
  MoveL 528 to (75.7, 19.21, 36) mm, rotated rx 180 ry 0 rz 180 deg; joints [-2.852, -2.09, -25.007, -172.709, -23.084, -6.713]
  MoveL 529 to (73.78, 25.77, 36) mm, rotated rx -180 ry 0 rz -180 deg; joints [-2.6, -2.203, -25.115, -173.348, -23.052, -6.125]
  MoveL 530 to (71.16, 32.28, 36) mm, rotated rx -180 ry 0 rz -180 deg; joints [-2.35, -2.348, -25.256, -173.981, -23.021, -5.542]
  MoveL 531 to (67.66, 39.11, 36) mm, rotated rx -180 ry 0 rz -180 deg; joints [-2.088, -2.537, -25.437, -174.648, -22.99, -4.929]
  MoveL 532 to (65.23, 42.94, 36) mm, rotated rx -180 ry 0 rz -180 deg; joints [-1.941, -2.667, -25.561, -175.021, -22.972, -4.586]
  MoveL 533 to (61.38, 48.38, 36) mm, rotated rx -180 ry 0 rz 180 deg; joints [-1.732, -2.869, -25.754, -175.555, -22.947, -4.095]
  MoveL 534 to (55.1, 55.43, 36) mm, rotated rx 180 ry 0 rz 180 deg; joints [-1.46, -3.196, -26.065, -176.248, -22.913, -3.457]
  MoveL 535 to (47.93, 61.73, 36) mm, rotated rx -180 ry 0 rz 180 deg; joints [-1.217, -3.565, -26.413, -176.869, -22.879, -2.885]
  MoveL 536 to (42.45, 65.57, 36) mm, rotated rx -180 ry 0 rz 180 deg; joints [-1.068, -3.846, -26.678, -177.25, -22.855, -2.534]
  MoveL 537 to (40.02, 67.13, 36) mm, rotated rx -180 ry 0 rz -180 deg; joints [-1.007, -3.97, -26.794, -177.404, -22.844, -2.392]
  MoveL 538 to (33.15, 70.78, 36) mm, rotated rx 180 ry 0 rz 180 deg; joints [-0.865, -4.322, -27.121, -177.768, -22.815, -2.058]
  MoveL 539 to (26.87, 73.39, 36) mm, rotated rx -180 ry 0 rz -180 deg; joints [-0.764, -4.642, -27.418, -178.028, -22.788, -1.818]
  MoveL 540 to (20.61, 75.35, 36) mm, rotated rx 180 ry 0 rz 180 deg; joints [-0.688, -4.962, -27.713, -178.222, -22.761, -1.639]
  MoveL 541 to (14.24, 76.85, 36) mm, rotated rx -180 ry 0 rz 180 deg; joints [-0.63, -5.287, -28.011, -178.37, -22.732, -1.503]
  MoveL 542 to (13.71, 76.94, 36) mm, rotated rx -180 ry 0 rz -180 deg; joints [-0.626, -5.314, -28.036, -178.38, -22.73, -1.495]
  MoveL 543 to (5.18, 77.98, 36) mm, rotated rx -180 ry 0 rz -180 deg; joints [-0.587, -5.75, -28.432, -178.477, -22.689, -1.405]
  MoveL 544 to (4.77, 78.01, 36) mm, rotated rx -180 ry 0 rz 180 deg; joints [-0.586, -5.771, -28.451, -178.48, -22.687, -1.403]
  MoveL 545 to (-2.78, 78.11, 36) mm, rotated rx 180 ry 0 rz 180 deg; joints [-0.585, -6.157, -28.799, -178.48, -22.65, -1.403]
  MoveL 546 to (-8.99, 77.62, 36) mm, rotated rx 180 ry 0 rz 180 deg; joints [-0.608, -6.475, -29.085, -178.419, -22.617, -1.46]
  MoveL 547 to (-16.39, 76.42, 36) mm, rotated rx -180 ry 0 rz -180 deg; joints [-0.662, -6.855, -29.423, -178.276, -22.578, -1.592]
  MoveL 548 to (-24.34, 74.26, 36) mm, rotated rx -180 ry 0 rz 180 deg; joints [-0.756, -7.262, -29.783, -178.027, -22.533, -1.822]
  MoveL 549 to (-32.49, 71.08, 36) mm, rotated rx -180 ry 0 rz -180 deg; joints [-0.895, -7.68, -30.15, -177.661, -22.487, -2.162]
  MoveL 550 to (-41.01, 66.53, 36) mm, rotated rx 180 ry 0 rz 180 deg; joints [-1.093, -8.116, -30.53, -177.135, -22.44, -2.648]
  MoveL 551 to (-44.27, 64.35, 36) mm, rotated rx 180 ry 0 rz 180 deg; joints [-1.189, -8.282, -30.674, -176.882, -22.422, -2.882]
  MoveL 552 to (-50.34, 59.77, 36) mm, rotated rx -180 ry 0 rz -180 deg; joints [-1.389, -8.592, -30.941, -176.35, -22.391, -3.375]
  MoveL 553 to (-55.98, 54.53, 36) mm, rotated rx -180 ry 0 rz -180 deg; joints [-1.62, -8.877, -31.186, -175.739, -22.365, -3.941]
  MoveL 554 to (-56.32, 54.18, 36) mm, rotated rx 180 ry 0 rz 180 deg; joints [-1.635, -8.895, -31.201, -175.698, -22.363, -3.979]
  MoveL 555 to (-60.68, 49.13, 36) mm, rotated rx 180 ry 0 rz 180 deg; joints [-1.858, -9.113, -31.388, -175.109, -22.348, -4.525]
  MoveL 556 to (-62.35, 47.13, 36) mm, rotated rx 180 ry 0 rz 180 deg; joints [-1.947, -9.196, -31.458, -174.873, -22.343, -4.744]
  MoveL 557 to (-67.52, 39.35, 36) mm, rotated rx 180 ry 0 rz 180 deg; joints [-2.29, -9.451, -31.674, -173.964, -22.335, -5.586]
  MoveL 558 to (-67.83, 38.82, 36) mm, rotated rx -180 ry 0 rz -180 deg; joints [-2.314, -9.466, -31.687, -173.901, -22.335, -5.645]
  MoveL 559 to (-71.98, 30.44, 36) mm, rotated rx -180 ry 0 rz 180 deg; joints [-2.684, -9.663, -31.854, -172.924, -22.344, -6.55]
  MoveL 560 to (-74.09, 24.8, 36) mm, rotated rx -180 ry 0 rz 180 deg; joints [-2.933, -9.759, -31.934, -172.268, -22.359, -7.157]
  MoveL 561 to (-75.11, 21.52, 36) mm, rotated rx 180 ry 0 rz 180 deg; joints [-3.078, -9.803, -31.971, -171.889, -22.37, -7.508]
  MoveL 562 to (-76.57, 15.64, 36) mm, rotated rx -180 ry 0 rz -180 deg; joints [-3.337, -9.862, -32.021, -171.212, -22.396, -8.134]
  MoveL 563 to (-77.49, 9.59, 36) mm, rotated rx -180 ry 0 rz 180 deg; joints [-3.602, -9.891, -32.045, -170.522, -22.431, -8.772]
  MoveL 564 to (-78.1, 2.95, 36) mm, rotated rx -180 ry 0 rz -180 deg; joints [-3.893, -9.9, -32.053, -169.771, -22.475, -9.466]
  MoveL 565 to (-78.03, -4.02, 36) mm, rotated rx -180 ry 0 rz -180 deg; joints [-4.195, -9.871, -32.028, -168.996, -22.531, -10.183]
  MoveL 566 to (-77.41, -10.72, 36) mm, rotated rx -180 ry 0 rz -180 deg; joints [-4.483, -9.812, -31.979, -168.261, -22.593, -10.861]
  MoveL 567 to (-76.37, -16.32, 36) mm, rotated rx 180 ry 0 rz 180 deg; joints [-4.722, -9.734, -31.914, -167.657, -22.652, -11.417]
  MoveL 568 to (-74.85, -22.35, 36) mm, rotated rx 180 ry 0 rz 180 deg; joints [-4.978, -9.629, -31.825, -167.017, -22.72, -12.006]
  MoveL 569 to (-73.44, -26.75, 36) mm, rotated rx -180 ry 0 rz 180 deg; joints [-5.162, -9.535, -31.745, -166.56, -22.773, -12.426]
  MoveL 570 to (-70.72, -33.22, 36) mm, rotated rx -180 ry 0 rz -180 deg; joints [-5.43, -9.362, -31.599, -165.9, -22.858, -13.032]
  MoveL 571 to (-67.72, -39.01, 36) mm, rotated rx -180 ry 0 rz 180 deg; joints [-5.666, -9.178, -31.442, -165.327, -22.939, -13.558]
  MoveL 572 to (-65.14, -43.06, 36) mm, rotated rx -180 ry 0 rz 180 deg; joints [-5.828, -9.023, -31.311, -164.936, -23, -13.915]
  MoveL 573 to (-61.42, -48.32, 36) mm, rotated rx -180 ry 0 rz -180 deg; joints [-6.036, -8.803, -31.122, -164.441, -23.081, -14.367]
  MoveL 574 to (-55.14, -55.39, 36) mm, rotated rx 180 ry 0 rz 180 deg; joints [-6.308, -8.439, -30.81, -163.806, -23.199, -14.946]
  MoveL 575 to (-48.36, -61.36, 36) mm, rotated rx -180 ry 0 rz -180 deg; joints [-6.528, -8.056, -30.478, -163.302, -23.306, -15.403]
  Set speed (16.7 mm/s)
  MoveL 576 to (-47.8, -61.63, 36) mm, rotated rx 180 ry 0 rz 180 deg; joints [-6.536, -8.025, -30.452, -163.283, -23.312, -15.42]
  MoveL 577 to (-47.18, -61.59, 36) mm, rotated rx -180 ry 0 rz -180 deg; joints [-6.532, -7.994, -30.424, -163.297, -23.315, -15.407]
  MoveL 578 to (-46.67, -61.25, 36) mm, rotated rx -180 ry 0 rz 180 deg; joints [-6.515, -7.969, -30.403, -163.34, -23.313, -15.367]
  MoveL 579 to (-46.77, -59.55, 36) mm, rotated rx -180 ry 0 rz 180 deg; joints [-6.444, -7.985, -30.416, -163.512, -23.293, -15.209]
  MoveL 580 to (-41.5, -52.51, 36) mm, rotated rx -180 ry 0 rz 180 deg; joints [-6.123, -7.753, -30.215, -164.315, -23.239, -14.468]
  Set speed (5.0 mm/s)
  MoveL 581 to (-41.5, -52.51, 30) mm, rotated rx -180 ry 0 rz -180 deg; joints [-6.123, -7.693, -30.442, -164.494, -23.516, -14.273]
  MoveL 582 to (-43.18, -52.72, 30) mm, rotated rx 180 ry 0 rz 180 deg; joints [-6.14, -7.778, -30.516, -164.447, -23.51, -14.317]
  MoveL 583 to (-43.42, -53.29, 30) mm, rotated rx -180 ry 0 rz -180 deg; joints [-6.165, -7.787, -30.524, -164.386, -23.515, -14.374]
  MoveL 584 to (-43.34, -53.91, 30) mm, rotated rx -180 ry 0 rz 180 deg; joints [-6.191, -7.78, -30.518, -164.324, -23.523, -14.43]
  MoveL 585 to (-42.97, -54.4, 30) mm, rotated rx 180 ry 0 rz 180 deg; joints [-6.21, -7.758, -30.499, -164.28, -23.53, -14.47]
  Set speed (16.7 mm/s)
  MoveL 586 to (-39.11, -57.4, 30) mm, rotated rx -180 ry 0 rz -180 deg; joints [-6.317, -7.543, -30.311, -164.036, -23.583, -14.691]
  MoveL 587 to (-34.51, -60.27, 30) mm, rotated rx -180 ry 0 rz -180 deg; joints [-6.416, -7.291, -30.089, -163.816, -23.637, -14.889]
  MoveL 588 to (-30.79, -62.23, 30) mm, rotated rx -180 ry 0 rz 180 deg; joints [-6.48, -7.089, -29.911, -163.677, -23.677, -15.013]
  MoveL 589 to (-24.49, -64.99, 30) mm, rotated rx 180 ry 0 rz 180 deg; joints [-6.565, -6.751, -29.611, -163.498, -23.735, -15.173]
  MoveL 590 to (-16.83, -67.38, 30) mm, rotated rx -180 ry 0 rz -180 deg; joints [-6.627, -6.346, -29.249, -163.378, -23.793, -15.278]
  MoveL 591 to (-11.44, -68.51, 30) mm, rotated rx 180 ry 0 rz 180 deg; joints [-6.647, -6.065, -28.997, -163.348, -23.826, -15.302]
  MoveL 592 to (-4.37, -69.32, 30) mm, rotated rx -180 ry 0 rz 180 deg; joints [-6.647, -5.701, -28.668, -163.372, -23.859, -15.276]
  MoveL 593 to (2.25, -69.37, 30) mm, rotated rx -180 ry 0 rz -180 deg; joints [-6.618, -5.365, -28.363, -163.461, -23.881, -15.191]
  MoveL 594 to (8.27, -68.96, 30) mm, rotated rx -180 ry 0 rz 180 deg; joints [-6.573, -5.062, -28.086, -163.584, -23.894, -15.076]
  MoveL 595 to (9.56, -68.75, 30) mm, rotated rx -180 ry 0 rz -180 deg; joints [-6.558, -4.999, -28.027, -163.622, -23.895, -15.04]
  MoveL 596 to (16.64, -67.43, 30) mm, rotated rx 180 ry 0 rz 180 deg; joints [-6.473, -4.649, -27.705, -163.844, -23.9, -14.835]
  MoveL 597 to (24.71, -64.91, 30) mm, rotated rx -180 ry 0 rz 180 deg; joints [-6.335, -4.255, -27.34, -164.19, -23.892, -14.515]
  MoveL 598 to (32.13, -61.58, 30) mm, rotated rx 180 ry 0 rz -180 deg; joints [-6.17, -3.9, -27.008, -164.6, -23.874, -14.138]
  MoveL 599 to (36.36, -59.17, 30) mm, rotated rx 180 ry 0 rz 180 deg; joints [-6.057, -3.7, -26.821, -164.879, -23.859, -13.881]
  MoveL 600 to (40.44, -56.45, 30) mm, rotated rx 180 ry 0 rz 180 deg; joints [-5.932, -3.509, -26.641, -165.186, -23.84, -13.599]
  MoveL 601 to (45.24, -52.7, 30) mm, rotated rx 180 ry 0 rz 180 deg; joints [-5.764, -3.287, -26.432, -165.597, -23.813, -13.222]
  MoveL 602 to (50.34, -47.85, 30) mm, rotated rx -180 ry 0 rz -180 deg; joints [-5.553, -3.055, -26.212, -166.114, -23.777, -12.748]
  MoveL 603 to (53.04, -44.84, 30) mm, rotated rx -180 ry 0 rz 180 deg; joints [-5.424, -2.934, -26.097, -166.429, -23.755, -12.459]
  MoveL 604 to (58.26, -37.82, 30) mm, rotated rx 180 ry 0 rz 180 deg; joints [-5.13, -2.705, -25.878, -167.15, -23.703, -11.798]
  MoveL 605 to (60.28, -34.49, 30) mm, rotated rx 180 ry 0 rz 180 deg; joints [-4.992, -2.618, -25.795, -167.487, -23.679, -11.489]
  MoveL 606 to (63.06, -29.12, 30) mm, rotated rx -180 ry 0 rz 180 deg; joints [-4.772, -2.502, -25.684, -168.026, -23.641, -10.995]
  MoveL 607 to (64.96, -24.55, 30) mm, rotated rx -180 ry 0 rz 180 deg; joints [-4.588, -2.425, -25.61, -168.48, -23.61, -10.579]
  MoveL 608 to (65.73, -22.1, 30) mm, rotated rx -180 ry 0 rz -180 deg; joints [-4.489, -2.397, -25.582, -168.722, -23.593, -10.356]
  MoveL 609 to (67.61, -15.76, 30) mm, rotated rx 180 ry 0 rz -180 deg; joints [-4.236, -2.326, -25.515, -169.346, -23.551, -9.784]
  MoveL 610 to (68.96, -8.21, 30) mm, rotated rx -180 ry 0 rz -180 deg; joints [-3.938, -2.285, -25.476, -170.085, -23.504, -9.107]
  MoveL 611 to (69.45, -0.92, 30) mm, rotated rx -180 ry 0 rz -180 deg; joints [-3.652, -2.285, -25.476, -170.795, -23.46, -8.456]
  MoveL 612 to (69, 7.59, 30) mm, rotated rx -180 ry 0 rz -180 deg; joints [-3.32, -2.334, -25.522, -171.62, -23.412, -7.699]
  MoveL 613 to (67.15, 17.65, 30) mm, rotated rx -180 ry 0 rz -180 deg; joints [-2.93, -2.455, -25.638, -172.592, -23.358, -6.807]
  MoveL 614 to (66.01, 21.6, 30) mm, rotated rx 180 ry 0 rz 180 deg; joints [-2.777, -2.522, -25.703, -172.974, -23.338, -6.456]
  MoveL 615 to (64.95, 24.58, 30) mm, rotated rx 180 ry 0 rz 180 deg; joints [-2.662, -2.582, -25.76, -173.262, -23.322, -6.192]
  MoveL 616 to (63.19, 28.62, 30) mm, rotated rx 180 ry 0 rz 180 deg; joints [-2.507, -2.68, -25.854, -173.652, -23.302, -5.834]
  MoveL 617 to (60.91, 33.26, 30) mm, rotated rx -180 ry 0 rz -180 deg; joints [-2.328, -2.804, -25.973, -174.101, -23.279, -5.422]
  MoveL 618 to (57.25, 39.31, 30) mm, rotated rx -180 ry 0 rz 180 deg; joints [-2.095, -3, -26.16, -174.686, -23.249, -4.884]
  MoveL 619 to (53.49, 44.3, 30) mm, rotated rx -180 ry 0 rz -180 deg; joints [-1.903, -3.199, -26.348, -175.17, -23.223, -4.44]
  MoveL 620 to (50.18, 47.91, 30) mm, rotated rx 180 ry 0 rz 180 deg; joints [-1.764, -3.372, -26.512, -175.52, -23.203, -4.119]
  MoveL 621 to (45.95, 52.08, 30) mm, rotated rx 180 ry 0 rz 180 deg; joints [-1.603, -3.592, -26.719, -175.925, -23.18, -3.747]
  MoveL 622 to (39.07, 57.42, 30) mm, rotated rx -180 ry 0 rz 180 deg; joints [-1.397, -3.947, -27.052, -176.445, -23.145, -3.269]
  MoveL 623 to (34.59, 60.23, 30) mm, rotated rx -180 ry 0 rz -180 deg; joints [-1.288, -4.178, -27.268, -176.718, -23.124, -3.019]
  MoveL 624 to (30.76, 62.25, 30) mm, rotated rx 180 ry 0 rz 180 deg; joints [-1.21, -4.374, -27.45, -176.914, -23.106, -2.839]
  MoveL 625 to (24.45, 65.01, 30) mm, rotated rx 180 ry 0 rz 180 deg; joints [-1.104, -4.697, -27.749, -177.182, -23.077, -2.593]
  MoveL 626 to (16.79, 67.39, 30) mm, rotated rx -180 ry 0 rz 180 deg; joints [-1.013, -5.089, -28.11, -177.411, -23.042, -2.383]
  MoveL 627 to (12.13, 68.39, 30) mm, rotated rx 180 ry 0 rz 180 deg; joints [-0.976, -5.327, -28.328, -177.504, -23.02, -2.298]
  MoveL 628 to (4.44, 69.31, 30) mm, rotated rx -180 ry 0 rz 180 deg; joints [-0.943, -5.721, -28.686, -177.584, -22.983, -2.225]
  MoveL 629 to (-2.28, 69.36, 30) mm, rotated rx 180 ry 0 rz 180 deg; joints [-0.946, -6.065, -28.997, -177.574, -22.95, -2.234]
  MoveL 630 to (-8.31, 68.96, 30) mm, rotated rx 180 ry 0 rz 180 deg; joints [-0.967, -6.373, -29.274, -177.517, -22.92, -2.287]
  MoveL 631 to (-9.59, 68.74, 30) mm, rotated rx 180 ry 0 rz 180 deg; joints [-0.977, -6.439, -29.332, -177.491, -22.913, -2.311]
  MoveL 632 to (-16.67, 67.43, 30) mm, rotated rx 180 ry 0 rz 180 deg; joints [-1.036, -6.801, -29.656, -177.333, -22.877, -2.457]
  MoveL 633 to (-24.74, 64.9, 30) mm, rotated rx -180 ry 0 rz -180 deg; joints [-1.149, -7.214, -30.021, -177.039, -22.835, -2.729]
  MoveL 634 to (-32.07, 61.61, 30) mm, rotated rx -180 ry 0 rz -180 deg; joints [-1.293, -7.588, -30.35, -176.66, -22.797, -3.079]
  MoveL 635 to (-36.3, 59.21, 30) mm, rotated rx 180 ry 0 rz 180 deg; joints [-1.399, -7.804, -30.539, -176.385, -22.776, -3.334]
  MoveL 636 to (-40.47, 56.42, 30) mm, rotated rx 180 ry 0 rz 180 deg; joints [-1.521, -8.015, -30.723, -176.065, -22.756, -3.63]
  MoveL 637 to (-45.27, 52.68, 30) mm, rotated rx 180 ry 0 rz 180 deg; joints [-1.686, -8.259, -30.934, -175.634, -22.735, -4.028]
  MoveL 638 to (-50.29, 47.91, 30) mm, rotated rx -180 ry 0 rz -180 deg; joints [-1.896, -8.511, -31.152, -175.085, -22.716, -4.535]
  MoveL 639 to (-52.99, 44.9, 30) mm, rotated rx 180 ry 0 rz 180 deg; joints [-2.028, -8.646, -31.268, -174.74, -22.708, -4.854]
  MoveL 640 to (-58.12, 38.01, 30) mm, rotated rx 180 ry 0 rz 180 deg; joints [-2.332, -8.899, -31.485, -173.948, -22.7, -5.586]
  MoveL 641 to (-60.31, 34.44, 30) mm, rotated rx 180 ry 0 rz 180 deg; joints [-2.489, -9.005, -31.575, -173.539, -22.7, -5.965]
  MoveL 642 to (-63.01, 29.22, 30) mm, rotated rx 180 ry 0 rz 180 deg; joints [-2.719, -9.133, -31.684, -172.941, -22.706, -6.517]
  MoveL 643 to (-64.99, 24.5, 30) mm, rotated rx 180 ry 0 rz 180 deg; joints [-2.926, -9.224, -31.762, -172.403, -22.717, -7.014]
  MoveL 644 to (-65.75, 22.03, 30) mm, rotated rx -180 ry 0 rz 180 deg; joints [-3.035, -9.257, -31.79, -172.124, -22.726, -7.272]
  MoveL 645 to (-67.63, 15.67, 30) mm, rotated rx 180 ry 0 rz 180 deg; joints [-3.313, -9.336, -31.857, -171.405, -22.751, -7.935]
  MoveL 646 to (-68.93, 8.4, 30) mm, rotated rx -180 ry 0 rz -180 deg; joints [-3.631, -9.381, -31.895, -170.591, -22.79, -8.686]
  MoveL 647 to (-68.98, 8.1, 30) mm, rotated rx -180 ry 0 rz 180 deg; joints [-3.643, -9.382, -31.896, -170.558, -22.792, -8.716]
  MoveL 648 to (-69.44, 1.23, 30) mm, rotated rx -180 ry 0 rz -180 deg; joints [-3.941, -9.383, -31.897, -169.8, -22.839, -9.415]
  MoveL 649 to (-68.98, -7.87, 30) mm, rotated rx -180 ry 0 rz -180 deg; joints [-4.332, -9.325, -31.847, -168.813, -22.914, -10.324]
  MoveL 650 to (-67.25, -17.3, 30) mm, rotated rx 180 ry 0 rz 180 deg; joints [-4.732, -9.196, -31.738, -167.816, -23.008, -11.241]
  MoveL 651 to (-65.02, -24.41, 30) mm, rotated rx -180 ry 0 rz 180 deg; joints [-5.029, -9.049, -31.613, -167.084, -23.089, -11.913]
  MoveL 652 to (-61.71, -31.87, 30) mm, rotated rx -180 ry 0 rz 180 deg; joints [-5.335, -8.842, -31.436, -166.338, -23.183, -12.596]
  MoveL 653 to (-60.96, -33.17, 30) mm, rotated rx -180 ry 0 rz -180 deg; joints [-5.388, -8.797, -31.398, -166.211, -23.201, -12.712]
  MoveL 654 to (-57.3, -39.25, 30) mm, rotated rx -180 ry 0 rz -180 deg; joints [-5.632, -8.577, -31.209, -165.626, -23.286, -13.246]
  MoveL 655 to (-53.4, -44.41, 30) mm, rotated rx 180 ry 0 rz 180 deg; joints [-5.835, -8.349, -31.012, -165.147, -23.364, -13.683]
  MoveL 656 to (-50.22, -47.87, 30) mm, rotated rx -180 ry 0 rz -180 deg; joints [-5.967, -8.167, -30.855, -164.838, -23.419, -13.964]
  MoveL 657 to (-45.87, -52.15, 30) mm, rotated rx 180 ry 0 rz 180 deg; joints [-6.128, -7.92, -30.64, -164.465, -23.49, -14.303]
  MoveL 658 to (-42.97, -54.4, 30) mm, rotated rx 180 ry 0 rz 180 deg; joints [-6.21, -7.758, -30.499, -164.28, -23.53, -14.47]
  Set speed (16.7 mm/s)
  MoveL 659 to (-42.4, -54.64, 30) mm, rotated rx -180 ry 0 rz -180 deg; joints [-6.217, -7.727, -30.472, -164.264, -23.536, -14.484]
  MoveL 660 to (-41.78, -54.57, 30) mm, rotated rx -180 ry 0 rz 180 deg; joints [-6.211, -7.696, -30.445, -164.281, -23.538, -14.468]
  MoveL 661 to (-41.29, -54.19, 30) mm, rotated rx -180 ry 0 rz -180 deg; joints [-6.193, -7.673, -30.424, -164.327, -23.536, -14.426]
  MoveL 662 to (-41.5, -52.5, 30) mm, rotated rx -180 ry 0 rz 180 deg; joints [-6.123, -7.693, -30.442, -164.494, -23.516, -14.273]
  Set speed (1000.0 mm/s)
  MoveL 663 to (-34.69, -44.49, 30) mm, rotated rx -180 ry 0 rz 180 deg; joints [-5.758, -7.386, -30.173, -165.407, -23.465, -13.432]
  Set speed (5.0 mm/s)
  MoveL 664 to (-34.69, -44.49, 24) mm, rotated rx 180 ry 0 rz 180 deg; joints [-5.758, -7.324, -30.398, -165.572, -23.744, -13.252]
  MoveL 665 to (-36.38, -44.64, 24) mm, rotated rx -180 ry 0 rz -180 deg; joints [-5.772, -7.41, -30.474, -165.533, -23.737, -13.288]
  MoveL 666 to (-36.64, -45.21, 24) mm, rotated rx -180 ry 0 rz 180 deg; joints [-5.796, -7.42, -30.483, -165.473, -23.742, -13.344]
  MoveL 667 to (-36.59, -45.83, 24) mm, rotated rx 180 ry 0 rz 180 deg; joints [-5.822, -7.414, -30.478, -165.411, -23.748, -13.4]
  MoveL 668 to (-36.23, -46.33, 24) mm, rotated rx -180 ry 0 rz -180 deg; joints [-5.842, -7.393, -30.46, -165.365, -23.755, -13.442]
  Set speed (16.7 mm/s)
  MoveL 669 to (-35.55, -46.9, 24) mm, rotated rx 180 ry 0 rz 180 deg; joints [-5.862, -7.356, -30.426, -165.318, -23.765, -13.485]
  MoveL 670 to (-31, -50.06, 24) mm, rotated rx -180 ry 0 rz 180 deg; joints [-5.975, -7.105, -30.206, -165.064, -23.82, -13.714]
  MoveL 671 to (-25.92, -52.8, 24) mm, rotated rx 180 ry 0 rz 180 deg; joints [-6.066, -6.83, -29.962, -164.862, -23.872, -13.895]
  MoveL 672 to (-22.38, -54.38, 24) mm, rotated rx 180 ry 0 rz 180 deg; joints [-6.116, -6.641, -29.793, -164.755, -23.904, -13.991]
  MoveL 673 to (-18.87, -55.74, 24) mm, rotated rx 180 ry 0 rz 180 deg; joints [-6.157, -6.454, -29.627, -164.67, -23.933, -14.067]
  MoveL 674 to (-15.53, -56.8, 24) mm, rotated rx 180 ry 0 rz -180 deg; joints [-6.186, -6.277, -29.469, -164.612, -23.958, -14.118]
  MoveL 675 to (-10.44, -57.92, 24) mm, rotated rx -180 ry 0 rz 180 deg; joints [-6.209, -6.012, -29.23, -164.573, -23.989, -14.151]
  MoveL 676 to (-5.95, -58.53, 24) mm, rotated rx 180 ry 0 rz 180 deg; joints [-6.214, -5.781, -29.021, -164.574, -24.012, -14.147]
  MoveL 677 to (-1.21, -58.88, 24) mm, rotated rx 180 ry 0 rz 180 deg; joints [-6.207, -5.538, -28.8, -164.604, -24.032, -14.118]
  MoveL 678 to (4.95, -58.68, 24) mm, rotated rx -180 ry 0 rz 180 deg; joints [-6.172, -5.226, -28.516, -164.704, -24.05, -14.023]
  MoveL 679 to (10.91, -57.87, 24) mm, rotated rx 180 ry 0 rz 180 deg; joints [-6.113, -4.929, -28.244, -164.859, -24.06, -13.879]
  MoveL 680 to (17.41, -56.2, 24) mm, rotated rx -180 ry 0 rz -180 deg; joints [-6.018, -4.609, -27.948, -165.099, -24.061, -13.657]
  MoveL 681 to (24.64, -53.49, 24) mm, rotated rx -180 ry 0 rz -180 deg; joints [-5.879, -4.258, -27.623, -165.446, -24.053, -13.337]
  MoveL 682 to (28.73, -51.41, 24) mm, rotated rx 180 ry 0 rz 180 deg; joints [-5.779, -4.062, -27.441, -165.692, -24.043, -13.111]
  MoveL 683 to (33.29, -48.58, 24) mm, rotated rx -180 ry 0 rz -180 deg; joints [-5.648, -3.846, -27.239, -166.013, -24.027, -12.816]
  MoveL 684 to (37.66, -45.27, 24) mm, rotated rx 180 ry 0 rz 180 deg; joints [-5.499, -3.642, -27.047, -166.377, -24.007, -12.484]
  MoveL 685 to (42.08, -41.11, 24) mm, rotated rx -180 ry 0 rz -180 deg; joints [-5.317, -3.439, -26.856, -166.819, -23.98, -12.078]
  MoveL 686 to (46.55, -36.08, 24) mm, rotated rx 180 ry 0 rz 180 deg; joints [-5.102, -3.238, -26.666, -167.343, -23.946, -11.598]
  MoveL 687 to (48.97, -32.7, 24) mm, rotated rx -180 ry 0 rz 180 deg; joints [-4.96, -3.131, -26.564, -167.689, -23.924, -11.282]
  MoveL 688 to (51.07, -29.19, 24) mm, rotated rx -180 ry 0 rz -180 deg; joints [-4.815, -3.04, -26.479, -168.043, -23.9, -10.957]
  MoveL 689 to (52.5, -26.46, 24) mm, rotated rx 180 ry 0 rz 180 deg; joints [-4.702, -2.98, -26.421, -168.318, -23.882, -10.706]
  MoveL 690 to (54.49, -22.34, 24) mm, rotated rx -180 ry 0 rz 180 deg; joints [-4.534, -2.897, -26.342, -168.729, -23.855, -10.33]
  MoveL 691 to (56.65, -15.86, 24) mm, rotated rx -180 ry 0 rz -180 deg; joints [-4.272, -2.813, -26.262, -169.369, -23.813, -9.744]
  MoveL 692 to (57.92, -10.62, 24) mm, rotated rx 180 ry 0 rz 180 deg; joints [-4.062, -2.769, -26.22, -169.882, -23.781, -9.274]
  MoveL 693 to (58.66, -4.73, 24) mm, rotated rx 180 ry 0 rz 180 deg; joints [-3.828, -2.752, -26.204, -170.455, -23.745, -8.75]
  MoveL 694 to (58.89, 0.11, 24) mm, rotated rx -180 ry 0 rz -180 deg; joints [-3.637, -2.756, -26.208, -170.925, -23.716, -8.32]
  MoveL 695 to (58.53, 6.44, 24) mm, rotated rx -180 ry 0 rz 180 deg; joints [-3.389, -2.794, -26.243, -171.536, -23.68, -7.761]
  MoveL 696 to (57.5, 12.58, 24) mm, rotated rx 180 ry 0 rz 180 deg; joints [-3.149, -2.863, -26.31, -172.127, -23.645, -7.219]
  MoveL 697 to (56.25, 17.18, 24) mm, rotated rx 180 ry 0 rz 180 deg; joints [-2.971, -2.939, -26.382, -172.568, -23.62, -6.815]
  MoveL 698 to (53.98, 23.4, 24) mm, rotated rx 180 ry 0 rz 180 deg; joints [-2.729, -3.068, -26.505, -173.166, -23.586, -6.268]
  MoveL 699 to (52.13, 27.4, 24) mm, rotated rx 180 ry 0 rz 180 deg; joints [-2.574, -3.171, -26.603, -173.549, -23.565, -5.917]
  MoveL 700 to (50.47, 30.32, 24) mm, rotated rx -180 ry 0 rz 180 deg; joints [-2.461, -3.261, -26.688, -173.829, -23.548, -5.661]
  MoveL 701 to (46.74, 35.65, 24) mm, rotated rx 180 ry 0 rz 180 deg; joints [-2.256, -3.461, -26.876, -174.339, -23.518, -5.193]
  MoveL 702 to (43.32, 39.9, 24) mm, rotated rx -180 ry 0 rz 180 deg; joints [-2.092, -3.642, -27.047, -174.746, -23.493, -4.82]
  MoveL 703 to (39.48, 43.62, 24) mm, rotated rx -180 ry 0 rz 180 deg; joints [-1.948, -3.843, -27.236, -175.103, -23.469, -4.494]
  MoveL 704 to (35.51, 46.93, 24) mm, rotated rx 180 ry 0 rz 180 deg; joints [-1.821, -4.049, -27.429, -175.419, -23.446, -4.204]
  MoveL 705 to (30.96, 50.09, 24) mm, rotated rx 180 ry 0 rz 180 deg; joints [-1.7, -4.285, -27.648, -175.72, -23.422, -3.928]
  MoveL 706 to (25.88, 52.82, 24) mm, rotated rx 180 ry 0 rz 180 deg; joints [-1.595, -4.547, -27.891, -175.979, -23.396, -3.691]
  MoveL 707 to (22.34, 54.4, 24) mm, rotated rx -180 ry 0 rz -180 deg; joints [-1.535, -4.729, -28.06, -176.128, -23.378, -3.555]
  MoveL 708 to (18.84, 55.76, 24) mm, rotated rx 180 ry 0 rz 180 deg; joints [-1.484, -4.909, -28.226, -176.254, -23.361, -3.439]
  MoveL 709 to (15.49, 56.82, 24) mm, rotated rx 180 ry 0 rz 180 deg; joints [-1.445, -5.081, -28.383, -176.352, -23.345, -3.35]
  MoveL 710 to (10.51, 57.91, 24) mm, rotated rx 180 ry 0 rz 180 deg; joints [-1.405, -5.336, -28.617, -176.448, -23.321, -3.262]
  MoveL 711 to (5.92, 58.53, 24) mm, rotated rx 180 ry 0 rz 180 deg; joints [-1.384, -5.571, -28.831, -176.498, -23.298, -3.217]
  MoveL 712 to (1.18, 58.88, 24) mm, rotated rx -180 ry 0 rz 180 deg; joints [-1.375, -5.814, -29.051, -176.52, -23.275, -3.198]
  MoveL 713 to (-2.27, 58.85, 24) mm, rotated rx -180 ry 0 rz -180 deg; joints [-1.379, -5.991, -29.211, -176.505, -23.259, -3.212]
  MoveL 714 to (-7.88, 58.36, 24) mm, rotated rx 180 ry 0 rz 180 deg; joints [-1.405, -6.277, -29.468, -176.435, -23.231, -3.276]
  MoveL 715 to (-14.16, 57.14, 24) mm, rotated rx -180 ry 0 rz 180 deg; joints [-1.462, -6.598, -29.755, -176.285, -23.201, -3.415]
  MoveL 716 to (-19.45, 55.48, 24) mm, rotated rx -180 ry 0 rz 180 deg; joints [-1.537, -6.868, -29.995, -176.092, -23.176, -3.594]
